LIN {X 0,Y 405.871,Z 975.986,A -85,B 0,C 180,E1 10185.137,E2 10185.137} C_VEL
LIN {X 0,Y 407.952,Z 961.068,A -85,B 0,C 180,E1 10190.645,E2 10190.645} C_VEL
LIN {X 0,Y 411.972,Z 940.342,A -85,B 0,C 180,E1 10196.169,E2 10196.169} C_VEL
LIN {X 0,Y 417.617,Z 915.19,A -85,B 0,C 180,E1 10201.176,E2 10201.176} C_VEL
LIN {X 0,Y 424.499,Z 886.002,A -85,B 0,C 180,E1 10205.579,E2 10205.579} C_VEL
LIN {X 0,Y 432.002,Z 852.461,A -85,B 0,C 180,E1 10209.402,E2 10209.402} C_VEL
LIN {X 0,Y 439.513,Z 814.318,A -85,B 0,C 180,E1 10212.598,E2 10212.598} C_VEL
LIN {X 0,Y 446.008,Z 773.682,A -85,B 0,C 180,E1 10214.978,E2 10214.978} C_VEL
LIN {X 0,Y 444.947,Z 768.035,A -85,B 0,C 180,E1 10215.473,E2 10215.473} C_VEL
LIN {X 0,Y 431.141,Z 737.427,A -85,B 0,C 180,E1 10219.164,E2 10219.164} C_VEL
LIN {X 0,Y 414.149,Z 709.31,A -85,B 0,C 180,E1 10223.192,E2 10223.192} C_VEL
LIN {X 0,Y 406.063,Z 697.489,A -85,B 0,C 180,E1 10225.147,E2 10225.147} C_VEL
LIN {X 0,Y 403.307,Z 692.479,A -85,B 0,C 180,E1 10225.876,E2 10225.876} C_VEL
LIN {X 0,Y 403.251,Z 691.44,A -85,B 0,C 180,E1 10226.097,E2 10226.097} C_VEL
LIN {X 0,Y 403.428,Z 691.44,A -85,B 0,C 180,E1 10233.243,E2 10233.243} C_VEL
LIN {X 0,Y 403.698,Z 691.44,A -85,B 0,C 180,E1 10240.281,E2 10240.281} C_VEL
LIN {X 0,Y 403.994,Z 691.44,A -85,B 0,C 180,E1 10247.012,E2 10247.012} C_VEL
LIN {X 0,Y 404.187,Z 691.44,A -85,B 0,C 180,E1 10253.554,E2 10253.554} C_VEL
LIN {X 0,Y 404.547,Z 691.44,A -85,B 0,C 180,E1 10260.005,E2 10260.005} C_VEL
LIN {X 0,Y 404.199,Z 691.44,A -85,B 0,C 180,E1 10266.457,E2 10266.457} C_VEL
LIN {X 0,Y 403.89,Z 691.44,A -85,B 0,C 180,E1 10273.002,E2 10273.002} C_VEL
LIN {X 0,Y 403.653,Z 691.44,A -85,B 0,C 180,E1 10279.732,E2 10279.732} C_VEL
LIN {X 0,Y 403.436,Z 691.44,A -85,B 0,C 180,E1 10286.768,E2 10286.768} C_VEL
LIN {X 0,Y 403.325,Z 692.074,A -85,B 0,C 180,E1 10293.543,E2 10293.543} C_VEL
LIN {X 0,Y 405.891,Z 697.335,A -85,B 0,C 180,E1 10294.241,E2 10294.241} C_VEL
LIN {X 0,Y 408.427,Z 700.839,A -85,B 0,C 180,E1 10294.859,E2 10294.859} C_VEL
LIN {X 0,Y 427.36,Z 729.308,A -85,B 0,C 180,E1 10299.089,E2 10299.089} C_VEL
LIN {X 0,Y 444.306,Z 761.012,A -85,B 0,C 180,E1 10302.797,E2 10302.797} C_VEL
LIN {X 0,Y 448.42,Z 772.307,A -85,B 0,C 180,E1 10303.868,E2 10303.868} C_VEL
LIN {X 0,Y 442.82,Z 814.858,A -85,B 0,C 180,E1 10305.797,E2 10305.797} C_VEL
LIN {X 0,Y 435.789,Z 854.926,A -85,B 0,C 180,E1 10308.487,E2 10308.487} C_VEL
LIN {X 0,Y 427.875,Z 893.059,A -85,B 0,C 180,E1 10312.061,E2 10312.061} C_VEL
LIN {X 0,Y 420.295,Z 927.543,A -85,B 0,C 180,E1 10316.454,E2 10316.454} C_VEL
LIN {X 0,Y 413.816,Z 957.71,A -85,B 0,C 180,E1 10321.599,E2 10321.599} C_VEL
LIN {X 0,Y 409.877,Z 978.091,A -85,B 0,C 180,E1 10326.142,E2 10326.142} C_VEL
LIN {X 0,Y 407.965,Z 982.373,A -85,B 0,C 180,E1 10327.183,E2 10327.183} C_VEL
LIN {X 0,Y 399.703,Z 993.008,A -85,B 0,C 180,E1 10330.043,E2 10330.043} C_VEL
LIN {X 0,Y 399.497,Z 993.911,A -85,B 0,C 180,E1 10330.327,E2 10330.327} C_VEL
LIN {X 0,Y 397.623,Z 1008.916,A -85,B 0,C 180,E1 10336.293,E2 10336.293} C_VEL
LIN {X 0,Y 397.001,Z 1017.213,A -85,B 0,C 180,E1 10341.226,E2 10341.226} C_VEL
LIN {X 0,Y 396.743,Z 1021.482,A -85,B 0,C 180,E1 10345.623,E2 10345.623} C_VEL
LIN {X 0,Y 396.752,Z 1022.899,A -85,B 0,C 180,E1 10350,E2 10350} C_VEL
LIN {X 0,Y 396.734,Z 1021.482,A -85,B 0,C 180,E1 10354.378,E2 10354.378} C_VEL
LIN {X 0,Y 397.07,Z 1015.608,A -85,B 0,C 180,E1 10359.881,E2 10359.881} C_VEL
LIN {X 0,Y 398.017,Z 1005.17,A -85,B 0,C 180,E1 10365.444,E2 10365.444} C_VEL
LIN {X 0,Y 400.499,Z 987.673,A -85,B 0,C 180,E1 10371.63,E2 10371.63} C_VEL
LIN {X 0,Y 405.041,Z 964.149,A -85,B 0,C 180,E1 10377.555,E2 10377.555} C_VEL
LIN {X 0,Y 411.393,Z 936.262,A -85,B 0,C 180,E1 10382.768,E2 10382.768} C_VEL
LIN {X 0,Y 419.069,Z 903.077,A -85,B 0,C 180,E1 10387.428,E2 10387.428} C_VEL
LIN {X 0,Y 427.424,Z 865.851,A -85,B 0,C 180,E1 10391.282,E2 10391.282} C_VEL
LIN {X 0,Y 435.091,Z 826.33,A -85,B 0,C 180,E1 10394.246,E2 10394.246} C_VEL
LIN {X 0,Y 441.567,Z 783.435,A -85,B 0,C 180,E1 10396.448,E2 10396.448} C_VEL
LIN {X 0,Y 442.358,Z 773.084,A -85,B 0,C 180,E1 10396.899,E2 10396.899} C_VEL
LIN {X 0,Y 427.471,Z 742.287,A -85,B 0,C 180,E1 10400.473,E2 10400.473} C_VEL
LIN {X 0,Y 410.7,Z 715.445,A -85,B 0,C 180,E1 10404.281,E2 10404.281} C_VEL
LIN {X 0,Y 398.509,Z 697.759,A -85,B 0,C 180,E1 10407.342,E2 10407.342} C_VEL
LIN {X 0,Y 395.501,Z 692.766,A -85,B 0,C 180,E1 10408.189,E2 10408.189} C_VEL
LIN {X 0,Y 395.382,Z 691.44,A -85,B 0,C 180,E1 10408.316,E2 10408.316} C_VEL
LIN {X 0,Y 395.521,Z 691.44,A -85,B 0,C 180,E1 10415.095,E2 10415.095} C_VEL
LIN {X 0,Y 395.755,Z 691.44,A -85,B 0,C 180,E1 10422.175,E2 10422.175} C_VEL
LIN {X 0,Y 395.918,Z 691.44,A -85,B 0,C 180,E1 10428.973,E2 10428.973} C_VEL
LIN {X 0,Y 396.325,Z 691.44,A -85,B 0,C 180,E1 10435.613,E2 10435.613} C_VEL
LIN {X 0,Y 396.584,Z 691.44,A -85,B 0,C 180,E1 10439.995,E2 10439.995} C_VEL
LIN {X 0,Y 396.272,Z 691.44,A -85,B 0,C 180,E1 10446.576,E2 10446.576} C_VEL
LIN {X 0,Y 395.972,Z 691.44,A -85,B 0,C 180,E1 10453.256,E2 10453.256} C_VEL
LIN {X 0,Y 395.763,Z 691.44,A -85,B 0,C 180,E1 10460.131,E2 10460.131} C_VEL
LIN {X 0,Y 395.465,Z 691.44,A -85,B 0,C 180,E1 10467.34,E2 10467.34} C_VEL
LIN {X 0,Y 395.414,Z 691.44,A -85,B 0,C 180,E1 10472.224,E2 10472.224} C_VEL
LIN {X 0,Y 397.431,Z 696.7,A -85,B 0,C 180,E1 10472.865,E2 10472.865} C_VEL
LIN {X 0,Y 400.544,Z 700.599,A -85,B 0,C 180,E1 10473.678,E2 10473.678} C_VEL
LIN {X 0,Y 416.344,Z 724.657,A -85,B 0,C 180,E1 10477.679,E2 10477.679} C_VEL
LIN {X 0,Y 431.961,Z 754.146,A -85,B 0,C 180,E1 10481.744,E2 10481.744} C_VEL
LIN {X 0,Y 440.414,Z 774.599,A -85,B 0,C 180,E1 10484.234,E2 10484.234} C_VEL
LIN {X 0,Y 433.168,Z 817.314,A -85,B 0,C 180,E1 10486.78,E2 10486.78} C_VEL
LIN {X 0,Y 425.102,Z 855.93,A -85,B 0,C 180,E1 10490.125,E2 10490.125} C_VEL
LIN {X 0,Y 417.01,Z 890.098,A -85,B 0,C 180,E1 10494.18,E2 10494.18} C_VEL
LIN {X 0,Y 409.351,Z 920.988,A -85,B 0,C 180,E1 10499.122,E2 10499.122} C_VEL
LIN {X 0,Y 403.241,Z 947.182,A -85,B 0,C 180,E1 10504.818,E2 10504.818} C_VEL
LIN {X 0,Y 399.451,Z 967.283,A -85,B 0,C 180,E1 10510.858,E2 10510.858} C_VEL
LIN {X 0,Y 397.531,Z 981.028,A -85,B 0,C 180,E1 10516.789,E2 10516.789} C_VEL
LIN {X 0,Y 396.87,Z 989.319,A -85,B 0,C 180,E1 10522.606,E2 10522.606} C_VEL
LIN {X 0,Y 396.723,Z 992.824,A -85,B 0,C 180,E1 10527.812,E2 10527.812} C_VEL
LIN {X 0,Y 396.715,Z 992.797,A -85,B 0,C 180,E1 10532.187,E2 10532.187} C_VEL
LIN {X 0,Y 396.85,Z 989.248,A -85,B 0,C 180,E1 10537.371,E2 10537.371} C_VEL
LIN {X 0,Y 397.582,Z 980.849,A -85,B 0,C 180,E1 10543.208,E2 10543.208} C_VEL
LIN {X 0,Y 399.731,Z 965.902,A -85,B 0,C 180,E1 10549.543,E2 10549.543} C_VEL
LIN {X 0,Y 403.525,Z 945.764,A -85,B 0,C 180,E1 10555.461,E2 10555.461} C_VEL
LIN {X 0,Y 409.55,Z 920.56,A -85,B 0,C 180,E1 10560.86,E2 10560.86} C_VEL
LIN {X 0,Y 417.157,Z 889.469,A -85,B 0,C 180,E1 10565.813,E2 10565.813} C_VEL
LIN {X 0,Y 425.282,Z 855.209,A -85,B 0,C 180,E1 10569.854,E2 10569.854} C_VEL
LIN {X 0,Y 433.349,Z 816.503,A -85,B 0,C 180,E1 10573.181,E2 10573.181} C_VEL
LIN {X 0,Y 440.244,Z 774.615,A -85,B 0,C 180,E1 10575.694,E2 10575.694} C_VEL
LIN {X 0,Y 427.49,Z 744.686,A -85,B 0,C 180,E1 10579.381,E2 10579.381} C_VEL
LIN {X 0,Y 410.721,Z 715.714,A -85,B 0,C 180,E1 10583.622,E2 10583.622} C_VEL
LIN {X 0,Y 398.207,Z 697.529,A -85,B 0,C 180,E1 10586.822,E2 10586.822} C_VEL
LIN {X 0,Y 395.46,Z 692.854,A -85,B 0,C 180,E1 10587.599,E2 10587.599} C_VEL
LIN {X 0,Y 395.322,Z 691.44,A -85,B 0,C 180,E1 10587.77,E2 10587.77} C_VEL
LIN {X 0,Y 395.539,Z 691.44,A -85,B 0,C 180,E1 10595.107,E2 10595.107} C_VEL
LIN {X 0,Y 395.888,Z 691.44,A -85,B 0,C 180,E1 10602.192,E2 10602.192} C_VEL
LIN {X 0,Y 396.138,Z 691.44,A -85,B 0,C 180,E1 10608.99,E2 10608.99} C_VEL
LIN {X 0,Y 396.441,Z 691.44,A -85,B 0,C 180,E1 10615.625,E2 10615.625} C_VEL
LIN {X 0,Y 396.615,Z 691.44,A -85,B 0,C 180,E1 10622.193,E2 10622.193} C_VEL
LIN {X 0,Y 396.164,Z 691.44,A -85,B 0,C 180,E1 10628.798,E2 10628.798} C_VEL
LIN {X 0,Y 395.869,Z 691.44,A -85,B 0,C 180,E1 10635.532,E2 10635.532} C_VEL
LIN {X 0,Y 395.623,Z 691.44,A -85,B 0,C 180,E1 10642.504,E2 10642.504} C_VEL
LIN {X 0,Y 395.397,Z 691.44,A -85,B 0,C 180,E1 10649.856,E2 10649.856} C_VEL
LIN {X 0,Y 395.38,Z 691.837,A -85,B 0,C 180,E1 10651.776,E2 10651.776} C_VEL
LIN {X 0,Y 397.682,Z 697.026,A -85,B 0,C 180,E1 10652.472,E2 10652.472} C_VEL
LIN {X 0,Y 400.23,Z 700.075,A -85,B 0,C 180,E1 10653.132,E2 10653.132} C_VEL
LIN {X 0,Y 420.31,Z 729.973,A -85,B 0,C 180,E1 10657.926,E2 10657.926} C_VEL
LIN {X 0,Y 437.407,Z 761.803,A -85,B 0,C 180,E1 10661.868,E2 10661.868} C_VEL
LIN {X 0,Y 442.611,Z 774.779,A -85,B 0,C 180,E1 10663.231,E2 10663.231} C_VEL
LIN {X 0,Y 436.936,Z 815.44,A -85,B 0,C 180,E1 10665.114,E2 10665.114} C_VEL
LIN {X 0,Y 429.605,Z 855.135,A -85,B 0,C 180,E1 10667.809,E2 10667.809} C_VEL
LIN {X 0,Y 421.323,Z 893.161,A -85,B 0,C 180,E1 10671.421,E2 10671.421} C_VEL
LIN {X 0,Y 413.286,Z 927.882,A -85,B 0,C 180,E1 10675.923,E2 10675.923} C_VEL
LIN {X 0,Y 406.574,Z 957.4,A -85,B 0,C 180,E1 10681.046,E2 10681.046} C_VEL
LIN {X 0,Y 401.645,Z 981.707,A -85,B 0,C 180,E1 10686.683,E2 10686.683} C_VEL
LIN {X 0,Y 399.497,Z 993.911,A -85,B 0,C 180,E1 10690.327,E2 10690.327} C_VEL
LIN {X 0,Y 396.338,Z 999.066,A -85,B 0,C 180,E1 10692.008,E2 10692.008} C_VEL
LIN {X 0,Y 390.178,Z 1005.669,A -85,B 0,C 180,E1 10694.591,E2 10694.591} C_VEL
LIN {X 0,Y 390.011,Z 1006.311,A -85,B 0,C 180,E1 10694.899,E2 10694.899} C_VEL
LIN {X 0,Y 389.097,Z 1016.913,A -85,B 0,C 180,E1 10701.046,E2 10701.046} C_VEL
LIN {X 0,Y 388.839,Z 1021.185,A -85,B 0,C 180,E1 10705.534,E2 10705.534} C_VEL
LIN {X 0,Y 388.883,Z 1022.604,A -85,B 0,C 180,E1 10710,E2 10710} C_VEL
LIN {X 0,Y 388.831,Z 1021.185,A -85,B 0,C 180,E1 10714.467,E2 10714.467} C_VEL
LIN {X 0,Y 389.187,Z 1015.307,A -85,B 0,C 180,E1 10720.083,E2 10720.083} C_VEL
LIN {X 0,Y 390.208,Z 1004.866,A -85,B 0,C 180,E1 10725.761,E2 10725.761} C_VEL
LIN {X 0,Y 392.769,Z 987.927,A -85,B 0,C 180,E1 10731.907,E2 10731.907} C_VEL
LIN {X 0,Y 397.603,Z 964.446,A -85,B 0,C 180,E1 10737.977,E2 10737.977} C_VEL
LIN {X 0,Y 404.532,Z 935.531,A -85,B 0,C 180,E1 10743.472,E2 10743.472} C_VEL
LIN {X 0,Y 412.644,Z 902.628,A -85,B 0,C 180,E1 10748.135,E2 10748.135} C_VEL
LIN {X 0,Y 421.305,Z 865.723,A -85,B 0,C 180,E1 10751.998,E2 10751.998} C_VEL
LIN {X 0,Y 429.393,Z 825.785,A -85,B 0,C 180,E1 10755.012,E2 10755.012} C_VEL
LIN {X 0,Y 436.114,Z 783.096,A -85,B 0,C 180,E1 10757.21,E2 10757.21} C_VEL
LIN {X 0,Y 436.335,Z 775.895,A -85,B 0,C 180,E1 10757.577,E2 10757.577} C_VEL
LIN {X 0,Y 422.102,Z 745.957,A -85,B 0,C 180,E1 10761.2,E2 10761.2} C_VEL
LIN {X 0,Y 404.297,Z 717.07,A -85,B 0,C 180,E1 10765.501,E2 10765.501} C_VEL
LIN {X 0,Y 394.117,Z 702.978,A -85,B 0,C 180,E1 10768.167,E2 10768.167} C_VEL
LIN {X 0,Y 390.792,Z 697.897,A -85,B 0,C 180,E1 10769.13,E2 10769.13} C_VEL
LIN {X 0,Y 387.726,Z 693.299,A -85,B 0,C 180,E1 10770.055,E2 10770.055} C_VEL
LIN {X 0,Y 387.494,Z 691.44,A -85,B 0,C 180,E1 10770.29,E2 10770.29} C_VEL
LIN {X 0,Y 387.666,Z 691.44,A -85,B 0,C 180,E1 10777.008,E2 10777.008} C_VEL
LIN {X 0,Y 387.84,Z 691.44,A -85,B 0,C 180,E1 10784.138,E2 10784.138} C_VEL
LIN {X 0,Y 388.185,Z 691.44,A -85,B 0,C 180,E1 10791.02,E2 10791.02} C_VEL
LIN {X 0,Y 388.714,Z 691.44,A -85,B 0,C 180,E1 10797.763,E2 10797.763} C_VEL
LIN {X 0,Y 388.477,Z 691.44,A -85,B 0,C 180,E1 10804.465,E2 10804.465} C_VEL
LIN {X 0,Y 388.114,Z 691.44,A -85,B 0,C 180,E1 10811.241,E2 10811.241} C_VEL
LIN {X 0,Y 387.896,Z 691.44,A -85,B 0,C 180,E1 10818.188,E2 10818.188} C_VEL
LIN {X 0,Y 387.566,Z 691.44,A -85,B 0,C 180,E1 10825.441,E2 10825.441} C_VEL
LIN {X 0,Y 387.513,Z 691.604,A -85,B 0,C 180,E1 10830.313,E2 10830.313} C_VEL
LIN {X 0,Y 389.444,Z 696.62,A -85,B 0,C 180,E1 10830.978,E2 10830.978} C_VEL
LIN {X 0,Y 392.499,Z 700,A -85,B 0,C 180,E1 10831.835,E2 10831.835} C_VEL
LIN {X 0,Y 409.2,Z 725.217,A -85,B 0,C 180,E1 10836.37,E2 10836.37} C_VEL
LIN {X 0,Y 424.361,Z 753.408,A -85,B 0,C 180,E1 10840.51,E2 10840.51} C_VEL
LIN {X 0,Y 434.373,Z 777.629,A -85,B 0,C 180,E1 10843.602,E2 10843.602} C_VEL
LIN {X 0,Y 427.137,Z 818.664,A -85,B 0,C 180,E1 10846.124,E2 10846.124} C_VEL
LIN {X 0,Y 418.893,Z 856.23,A -85,B 0,C 180,E1 10849.412,E2 10849.412} C_VEL
LIN {X 0,Y 410.389,Z 890.63,A -85,B 0,C 180,E1 10853.549,E2 10853.549} C_VEL
LIN {X 0,Y 402.372,Z 921.29,A -85,B 0,C 180,E1 10858.526,E2 10858.526} C_VEL
LIN {X 0,Y 396.111,Z 946.646,A -85,B 0,C 180,E1 10864.093,E2 10864.093} C_VEL
LIN {X 0,Y 391.859,Z 967.323,A -85,B 0,C 180,E1 10870.37,E2 10870.37} C_VEL
LIN {X 0,Y 389.739,Z 981.327,A -85,B 0,C 180,E1 10876.52,E2 10876.52} C_VEL
LIN {X 0,Y 388.984,Z 989.616,A -85,B 0,C 180,E1 10882.455,E2 10882.455} C_VEL
LIN {X 0,Y 388.83,Z 993.12,A -85,B 0,C 180,E1 10887.768,E2 10887.768} C_VEL
LIN {X 0,Y 388.82,Z 993.094,A -85,B 0,C 180,E1 10892.231,E2 10892.231} C_VEL
LIN {X 0,Y 388.964,Z 989.547,A -85,B 0,C 180,E1 10897.521,E2 10897.521} C_VEL
LIN {X 0,Y 389.798,Z 981.15,A -85,B 0,C 180,E1 10903.477,E2 10903.477} C_VEL
LIN {X 0,Y 391.954,Z 967.034,A -85,B 0,C 180,E1 10909.648,E2 10909.648} C_VEL
LIN {X 0,Y 396.14,Z 946.287,A -85,B 0,C 180,E1 10915.915,E2 10915.915} C_VEL
LIN {X 0,Y 402.524,Z 920.874,A -85,B 0,C 180,E1 10921.459,E2 10921.459} C_VEL
LIN {X 0,Y 410.549,Z 890.02,A -85,B 0,C 180,E1 10926.443,E2 10926.443} C_VEL
LIN {X 0,Y 419.131,Z 855.517,A -85,B 0,C 180,E1 10930.559,E2 10930.559} C_VEL
LIN {X 0,Y 427.707,Z 816.033,A -85,B 0,C 180,E1 10933.967,E2 10933.967} C_VEL
LIN {X 0,Y 434.276,Z 777.765,A -85,B 0,C 180,E1 10936.306,E2 10936.306} C_VEL
LIN {X 0,Y 421.778,Z 747.945,A -85,B 0,C 180,E1 10940.144,E2 10940.144} C_VEL
LIN {X 0,Y 406.249,Z 720.645,A -85,B 0,C 180,E1 10944.315,E2 10944.315} C_VEL
LIN {X 0,Y 394.627,Z 703.593,A -85,B 0,C 180,E1 10947.432,E2 10947.432} C_VEL
LIN {X 0,Y 390.66,Z 697.774,A -85,B 0,C 180,E1 10948.567,E2 10948.567} C_VEL
LIN {X 0,Y 387.611,Z 692.986,A -85,B 0,C 180,E1 10949.493,E2 10949.493} C_VEL
LIN {X 0,Y 387.439,Z 691.44,A -85,B 0,C 180,E1 10949.682,E2 10949.682} C_VEL
LIN {X 0,Y 387.675,Z 691.44,A -85,B 0,C 180,E1 10957.02,E2 10957.02} C_VEL
LIN {X 0,Y 388.036,Z 691.44,A -85,B 0,C 180,E1 10964.157,E2 10964.157} C_VEL
LIN {X 0,Y 388.261,Z 691.44,A -85,B 0,C 180,E1 10971.233,E2 10971.233} C_VEL
LIN {X 0,Y 388.66,Z 691.44,A -85,B 0,C 180,E1 10977.773,E2 10977.773} C_VEL
LIN {X 0,Y 388.721,Z 691.44,A -85,B 0,C 180,E1 10982.237,E2 10982.237} C_VEL
LIN {X 0,Y 388.225,Z 691.44,A -85,B 0,C 180,E1 10988.979,E2 10988.979} C_VEL
LIN {X 0,Y 387.956,Z 691.44,A -85,B 0,C 180,E1 10995.858,E2 10995.858} C_VEL
LIN {X 0,Y 387.676,Z 691.44,A -85,B 0,C 180,E1 11002.991,E2 11002.991} C_VEL
LIN {X 0,Y 387.509,Z 691.752,A -85,B 0,C 180,E1 11009.864,E2 11009.864} C_VEL
LIN {X 0,Y 389.61,Z 696.874,A -85,B 0,C 180,E1 11010.572,E2 11010.572} C_VEL
LIN {X 0,Y 392.432,Z 699.946,A -85,B 0,C 180,E1 11011.36,E2 11011.36} C_VEL
LIN {X 0,Y 410.252,Z 726.239,A -85,B 0,C 180,E1 11015.98,E2 11015.98} C_VEL
LIN {X 0,Y 426.337,Z 753.807,A -85,B 0,C 180,E1 11019.818,E2 11019.818} C_VEL
LIN {X 0,Y 436.774,Z 777.147,A -85,B 0,C 180,E1 11022.559,E2 11022.559} C_VEL
LIN {X 0,Y 430.955,Z 816.904,A -85,B 0,C 180,E1 11024.464,E2 11024.464} C_VEL
LIN {X 0,Y 423.306,Z 856.219,A -85,B 0,C 180,E1 11027.189,E2 11027.189} C_VEL
LIN {X 0,Y 414.761,Z 893.451,A -85,B 0,C 180,E1 11030.781,E2 11030.781} C_VEL
LIN {X 0,Y 406.466,Z 927.503,A -85,B 0,C 180,E1 11035.258,E2 11035.258} C_VEL
LIN {X 0,Y 399.337,Z 957.089,A -85,B 0,C 180,E1 11040.47,E2 11040.47} C_VEL
LIN {X 0,Y 394.118,Z 981.399,A -85,B 0,C 180,E1 11046.211,E2 11046.211} C_VEL
LIN {X 0,Y 390.795,Z 1000.752,A -85,B 0,C 180,E1 11052.527,E2 11052.527} C_VEL
LIN {X 0,Y 390.011,Z 1006.311,A -85,B 0,C 180,E1 11054.899,E2 11054.899} C_VEL
LIN {X 0,Y 387.127,Z 1010.096,A -85,B 0,C 180,E1 11056.708,E2 11056.708} C_VEL
LIN {X 0,Y 381.403,Z 1014.666,A -85,B 0,C 180,E1 11059.46,E2 11059.46} C_VEL
LIN {X 0,Y 381.271,Z 1015.113,A -85,B 0,C 180,E1 11059.783,E2 11059.783} C_VEL
LIN {X 0,Y 380.936,Z 1020.888,A -85,B 0,C 180,E1 11065.441,E2 11065.441} C_VEL
LIN {X 0,Y 380.987,Z 1022.308,A -85,B 0,C 180,E1 11070,E2 11070} C_VEL
LIN {X 0,Y 380.927,Z 1020.888,A -85,B 0,C 180,E1 11074.56,E2 11074.56} C_VEL
LIN {X 0,Y 381.312,Z 1015.007,A -85,B 0,C 180,E1 11080.293,E2 11080.293} C_VEL
LIN {X 0,Y 382.409,Z 1004.561,A -85,B 0,C 180,E1 11086.091,E2 11086.091} C_VEL
LIN {X 0,Y 385.08,Z 988,A -85,B 0,C 180,E1 11092.241,E2 11092.241} C_VEL
LIN {X 0,Y 390.246,Z 964.424,A -85,B 0,C 180,E1 11098.483,E2 11098.483} C_VEL
LIN {X 0,Y 397.61,Z 935.371,A -85,B 0,C 180,E1 11104.106,E2 11104.106} C_VEL
LIN {X 0,Y 406.391,Z 901.628,A -85,B 0,C 180,E1 11108.933,E2 11108.933} C_VEL
LIN {X 0,Y 415.124,Z 866.198,A -85,B 0,C 180,E1 11112.681,E2 11112.681} C_VEL
LIN {X 0,Y 423.372,Z 827.365,A -85,B 0,C 180,E1 11115.664,E2 11115.664} C_VEL
LIN {X 0,Y 430.534,Z 784.272,A -85,B 0,C 180,E1 11117.93,E2 11117.93} C_VEL
LIN {X 0,Y 430.282,Z 778.38,A -85,B 0,C 180,E1 11118.306,E2 11118.306} C_VEL
LIN {X 0,Y 416.342,Z 748.795,A -85,B 0,C 180,E1 11122.061,E2 11122.061} C_VEL
LIN {X 0,Y 399.171,Z 720.875,A -85,B 0,C 180,E1 11126.456,E2 11126.456} C_VEL
LIN {X 0,Y 387.074,Z 703.849,A -85,B 0,C 180,E1 11129.84,E2 11129.84} C_VEL
LIN {X 0,Y 383.005,Z 697.964,A -85,B 0,C 180,E1 11131.115,E2 11131.115} C_VEL
LIN {X 0,Y 379.872,Z 693.418,A -85,B 0,C 180,E1 11132.153,E2 11132.153} C_VEL
LIN {X 0,Y 379.605,Z 691.44,A -85,B 0,C 180,E1 11132.374,E2 11132.374} C_VEL
LIN {X 0,Y 379.797,Z 691.44,A -85,B 0,C 180,E1 11138.971,E2 11138.971} C_VEL
LIN {X 0,Y 379.931,Z 691.44,A -85,B 0,C 180,E1 11146.162,E2 11146.162} C_VEL
LIN {X 0,Y 380.438,Z 691.44,A -85,B 0,C 180,E1 11153.138,E2 11153.138} C_VEL
LIN {X 0,Y 380.79,Z 691.44,A -85,B 0,C 180,E1 11159.994,E2 11159.994} C_VEL
LIN {X 0,Y 380.437,Z 691.44,A -85,B 0,C 180,E1 11166.851,E2 11166.851} C_VEL
LIN {X 0,Y 380.102,Z 691.44,A -85,B 0,C 180,E1 11173.82,E2 11173.82} C_VEL
LIN {X 0,Y 379.827,Z 691.44,A -85,B 0,C 180,E1 11181.015,E2 11181.015} C_VEL
LIN {X 0,Y 379.654,Z 691.44,A -85,B 0,C 180,E1 11188.175,E2 11188.175} C_VEL
LIN {X 0,Y 381.526,Z 696.61,A -85,B 0,C 180,E1 11188.915,E2 11188.915} C_VEL
LIN {X 0,Y 384.734,Z 700.036,A -85,B 0,C 180,E1 11189.903,E2 11189.903} C_VEL
LIN {X 0,Y 401.207,Z 724.075,A -85,B 0,C 180,E1 11194.711,E2 11194.711} C_VEL
LIN {X 0,Y 417.592,Z 754.476,A -85,B 0,C 180,E1 11199.454,E2 11199.454} C_VEL
LIN {X 0,Y 428.42,Z 780.825,A -85,B 0,C 180,E1 11202.984,E2 11202.984} C_VEL
LIN {X 0,Y 421.258,Z 819.645,A -85,B 0,C 180,E1 11205.424,E2 11205.424} C_VEL
LIN {X 0,Y 412.809,Z 856.527,A -85,B 0,C 180,E1 11208.685,E2 11208.685} C_VEL
LIN {X 0,Y 403.874,Z 891.026,A -85,B 0,C 180,E1 11212.88,E2 11212.88} C_VEL
LIN {X 0,Y 395.428,Z 921.593,A -85,B 0,C 180,E1 11217.908,E2 11217.908} C_VEL
LIN {X 0,Y 388.827,Z 946.909,A -85,B 0,C 180,E1 11223.559,E2 11223.559} C_VEL
LIN {X 0,Y 384.285,Z 967.226,A -85,B 0,C 180,E1 11229.807,E2 11229.807} C_VEL
LIN {X 0,Y 381.946,Z 981.626,A -85,B 0,C 180,E1 11236.24,E2 11236.24} C_VEL
LIN {X 0,Y 381.12,Z 989.616,A -85,B 0,C 180,E1 11242.007,E2 11242.007} C_VEL
LIN {X 0,Y 380.931,Z 993.416,A -85,B 0,C 180,E1 11247.722,E2 11247.722} C_VEL
LIN {X 0,Y 380.92,Z 993.39,A -85,B 0,C 180,E1 11252.278,E2 11252.278} C_VEL
LIN {X 0,Y 381.106,Z 989.524,A -85,B 0,C 180,E1 11257.992,E2 11257.992} C_VEL
LIN {X 0,Y 382.127,Z 980.528,A -85,B 0,C 180,E1 11264.237,E2 11264.237} C_VEL
LIN {X 0,Y 384.349,Z 966.958,A -85,B 0,C 180,E1 11270.201,E2 11270.201} C_VEL
LIN {X 0,Y 388.865,Z 946.539,A -85,B 0,C 180,E1 11276.452,E2 11276.452} C_VEL
LIN {X 0,Y 395.553,Z 921.183,A -85,B 0,C 180,E1 11282.08,E2 11282.08} C_VEL
LIN {X 0,Y 404.058,Z 890.442,A -85,B 0,C 180,E1 11287.107,E2 11287.107} C_VEL
LIN {X 0,Y 413.042,Z 855.824,A -85,B 0,C 180,E1 11291.286,E2 11291.286} C_VEL
LIN {X 0,Y 421.819,Z 817.265,A -85,B 0,C 180,E1 11294.655,E2 11294.655} C_VEL
LIN {X 0,Y 428.325,Z 780.971,A -85,B 0,C 180,E1 11296.923,E2 11296.923} C_VEL
LIN {X 0,Y 416.664,Z 752.449,A -85,B 0,C 180,E1 11300.732,E2 11300.732} C_VEL
LIN {X 0,Y 400.891,Z 723.831,A -85,B 0,C 180,E1 11305.258,E2 11305.258} C_VEL
LIN {X 0,Y 387.309,Z 704.154,A -85,B 0,C 180,E1 11309.168,E2 11309.168} C_VEL
LIN {X 0,Y 382.938,Z 697.914,A -85,B 0,C 180,E1 11310.53,E2 11310.53} C_VEL
LIN {X 0,Y 379.762,Z 693.059,A -85,B 0,C 180,E1 11311.59,E2 11311.59} C_VEL
LIN {X 0,Y 379.593,Z 691.44,A -85,B 0,C 180,E1 11311.739,E2 11311.739} C_VEL
LIN {X 0,Y 379.827,Z 691.44,A -85,B 0,C 180,E1 11318.985,E2 11318.985} C_VEL
LIN {X 0,Y 380.163,Z 691.44,A -85,B 0,C 180,E1 11326.182,E2 11326.182} C_VEL
LIN {X 0,Y 380.469,Z 691.44,A -85,B 0,C 180,E1 11333.15,E2 11333.15} C_VEL
LIN {X 0,Y 380.849,Z 691.44,A -85,B 0,C 180,E1 11340.006,E2 11340.006} C_VEL
LIN {X 0,Y 380.437,Z 691.44,A -85,B 0,C 180,E1 11346.862,E2 11346.862} C_VEL
LIN {X 0,Y 380.084,Z 691.44,A -85,B 0,C 180,E1 11353.832,E2 11353.832} C_VEL
LIN {X 0,Y 379.797,Z 691.44,A -85,B 0,C 180,E1 11361.029,E2 11361.029} C_VEL
LIN {X 0,Y 379.679,Z 692.237,A -85,B 0,C 180,E1 11367.782,E2 11367.782} C_VEL
LIN {X 0,Y 382.284,Z 697.399,A -85,B 0,C 180,E1 11368.702,E2 11368.702} C_VEL
LIN {X 0,Y 384.769,Z 700.188,A -85,B 0,C 180,E1 11369.466,E2 11369.466} C_VEL
LIN {X 0,Y 402.141,Z 725.186,A -85,B 0,C 180,E1 11374.338,E2 11374.338} C_VEL
LIN {X 0,Y 418.613,Z 753.04,A -85,B 0,C 180,E1 11378.52,E2 11378.52} C_VEL
LIN {X 0,Y 431.025,Z 780.4,A -85,B 0,C 180,E1 11381.924,E2 11381.924} C_VEL
LIN {X 0,Y 424.703,Z 820.098,A -85,B 0,C 180,E1 11383.898,E2 11383.898} C_VEL
LIN {X 0,Y 416.988,Z 857.539,A -85,B 0,C 180,E1 11386.568,E2 11386.568} C_VEL
LIN {X 0,Y 408.27,Z 893.853,A -85,B 0,C 180,E1 11390.139,E2 11390.139} C_VEL
LIN {X 0,Y 399.626,Z 927.5,A -85,B 0,C 180,E1 11394.632,E2 11394.632} C_VEL
LIN {X 0,Y 392.191,Z 956.779,A -85,B 0,C 180,E1 11399.876,E2 11399.876} C_VEL
LIN {X 0,Y 386.55,Z 981.089,A -85,B 0,C 180,E1 11405.715,E2 11405.715} C_VEL
LIN {X 0,Y 383.06,Z 1000.447,A -85,B 0,C 180,E1 11412.162,E2 11412.162} C_VEL
LIN {X 0,Y 381.402,Z 1013.369,A -85,B 0,C 180,E1 11418.552,E2 11418.552} C_VEL
LIN {X 0,Y 381.271,Z 1015.113,A -85,B 0,C 180,E1 11419.783,E2 11419.783} C_VEL
LIN {X 0,Y 378.543,Z 1017.527,A -85,B 0,C 180,E1 11421.689,E2 11421.689} C_VEL
LIN {X 0,Y 373.113,Z 1020.025,A -85,B 0,C 180,E1 11424.585,E2 11424.585} C_VEL
LIN {X 0,Y 373.033,Z 1020.27,A -85,B 0,C 180,E1 11424.921,E2 11424.921} C_VEL
LIN {X 0,Y 373.116,Z 1022.013,A -85,B 0,C 180,E1 11430,E2 11430} C_VEL
LIN {X 0,Y 373.053,Z 1020.592,A -85,B 0,C 180,E1 11434.656,E2 11434.656} C_VEL
LIN {X 0,Y 373.435,Z 1014.707,A -85,B 0,C 180,E1 11440.513,E2 11440.513} C_VEL
LIN {X 0,Y 374.615,Z 1004.257,A -85,B 0,C 180,E1 11446.435,E2 11446.435} C_VEL
LIN {X 0,Y 377.774,Z 986.506,A -85,B 0,C 180,E1 11453.079,E2 11453.079} C_VEL
LIN {X 0,Y 383.001,Z 964.061,A -85,B 0,C 180,E1 11459.086,E2 11459.086} C_VEL
LIN {X 0,Y 390.905,Z 934.708,A -85,B 0,C 180,E1 11464.842,E2 11464.842} C_VEL
LIN {X 0,Y 400.054,Z 901.322,A -85,B 0,C 180,E1 11469.67,E2 11469.67} C_VEL
LIN {X 0,Y 409.368,Z 865.116,A -85,B 0,C 180,E1 11473.521,E2 11473.521} C_VEL
LIN {X 0,Y 418.101,Z 825.607,A -85,B 0,C 180,E1 11476.546,E2 11476.546} C_VEL
LIN {X 0,Y 424.913,Z 782.579,A -85,B 0,C 180,E1 11478.862,E2 11478.862} C_VEL
LIN {X 0,Y 410.894,Z 752.103,A -85,B 0,C 180,E1 11482.886,E2 11482.886} C_VEL
LIN {X 0,Y 393.642,Z 723.678,A -85,B 0,C 180,E1 11487.575,E2 11487.575} C_VEL
LIN {X 0,Y 379.978,Z 704.567,A -85,B 0,C 180,E1 11491.688,E2 11491.688} C_VEL
LIN {X 0,Y 375.6,Z 698.26,A -85,B 0,C 180,E1 11493.199,E2 11493.199} C_VEL
LIN {X 0,Y 371.973,Z 693.472,A -85,B 0,C 180,E1 11494.523,E2 11494.523} C_VEL
LIN {X 0,Y 371.693,Z 691.44,A -85,B 0,C 180,E1 11494.836,E2 11494.836} C_VEL
LIN {X 0,Y 371.926,Z 691.44,A -85,B 0,C 180,E1 11500.99,E2 11500.99} C_VEL
LIN {X 0,Y 372.104,Z 691.44,A -85,B 0,C 180,E1 11508.257,E2 11508.257} C_VEL
LIN {X 0,Y 372.602,Z 691.44,A -85,B 0,C 180,E1 11515.333,E2 11515.333} C_VEL
LIN {X 0,Y 372.889,Z 691.44,A -85,B 0,C 180,E1 11519.994,E2 11519.994} C_VEL
LIN {X 0,Y 372.51,Z 691.44,A -85,B 0,C 180,E1 11526.997,E2 11526.997} C_VEL
LIN {X 0,Y 372.159,Z 691.44,A -85,B 0,C 180,E1 11534.121,E2 11534.121} C_VEL
LIN {X 0,Y 371.851,Z 691.44,A -85,B 0,C 180,E1 11541.488,E2 11541.488} C_VEL
LIN {X 0,Y 371.777,Z 692.123,A -85,B 0,C 180,E1 11545.838,E2 11545.838} C_VEL
LIN {X 0,Y 374.22,Z 697.201,A -85,B 0,C 180,E1 11546.822,E2 11546.822} C_VEL
LIN {X 0,Y 376.998,Z 699.956,A -85,B 0,C 180,E1 11547.765,E2 11547.765} C_VEL
LIN {X 0,Y 391.99,Z 721.692,A -85,B 0,C 180,E1 11552.56,E2 11552.56} C_VEL
LIN {X 0,Y 406.986,Z 747.516,A -85,B 0,C 180,E1 11557.11,E2 11557.11} C_VEL
LIN {X 0,Y 420.206,Z 777.379,A -85,B 0,C 180,E1 11561.452,E2 11561.452} C_VEL
LIN {X 0,Y 422.569,Z 784.223,A -85,B 0,C 180,E1 11562.371,E2 11562.371} C_VEL
LIN {X 0,Y 414.915,Z 823.042,A -85,B 0,C 180,E1 11564.895,E2 11564.895} C_VEL
LIN {X 0,Y 406.125,Z 859.23,A -85,B 0,C 180,E1 11568.196,E2 11568.196} C_VEL
LIN {X 0,Y 396.994,Z 892.805,A -85,B 0,C 180,E1 11572.394,E2 11572.394} C_VEL
LIN {X 0,Y 388.545,Z 921.896,A -85,B 0,C 180,E1 11577.269,E2 11577.269} C_VEL
LIN {X 0,Y 381.545,Z 947.212,A -85,B 0,C 180,E1 11583.014,E2 11583.014} C_VEL
LIN {X 0,Y 376.635,Z 967.596,A -85,B 0,C 180,E1 11589.405,E2 11589.405} C_VEL
LIN {X 0,Y 374.167,Z 981.924,A -85,B 0,C 180,E1 11595.948,E2 11595.948} C_VEL
LIN {X 0,Y 373.243,Z 989.913,A -85,B 0,C 180,E1 11601.837,E2 11601.837} C_VEL
LIN {X 0,Y 373.032,Z 993.712,A -85,B 0,C 180,E1 11607.673,E2 11607.673} C_VEL
LIN {X 0,Y 373.019,Z 993.687,A -85,B 0,C 180,E1 11612.326,E2 11612.326} C_VEL
LIN {X 0,Y 373.229,Z 989.824,A -85,B 0,C 180,E1 11618.162,E2 11618.162} C_VEL
LIN {X 0,Y 374.235,Z 981.755,A -85,B 0,C 180,E1 11624.048,E2 11624.048} C_VEL
LIN {X 0,Y 376.689,Z 967.371,A -85,B 0,C 180,E1 11630.591,E2 11630.591} C_VEL
LIN {X 0,Y 381.593,Z 946.847,A -85,B 0,C 180,E1 11636.996,E2 11636.996} C_VEL
LIN {X 0,Y 388.671,Z 921.492,A -85,B 0,C 180,E1 11642.718,E2 11642.718} C_VEL
LIN {X 0,Y 397.547,Z 890.981,A -85,B 0,C 180,E1 11647.781,E2 11647.781} C_VEL
LIN {X 0,Y 407.056,Z 856.13,A -85,B 0,C 180,E1 11652.03,E2 11652.03} C_VEL
LIN {X 0,Y 416.052,Z 818.109,A -85,B 0,C 180,E1 11655.39,E2 11655.39} C_VEL
LIN {X 0,Y 422.337,Z 783.871,A -85,B 0,C 180,E1 11657.595,E2 11657.595} C_VEL
LIN {X 0,Y 410.385,Z 754.28,A -85,B 0,C 180,E1 11661.722,E2 11661.722} C_VEL
LIN {X 0,Y 395.345,Z 727.262,A -85,B 0,C 180,E1 11666.279,E2 11666.279} C_VEL
LIN {X 0,Y 380.649,Z 705.15,A -85,B 0,C 180,E1 11670.875,E2 11670.875} C_VEL
LIN {X 0,Y 375.521,Z 698.192,A -85,B 0,C 180,E1 11672.614,E2 11672.614} C_VEL
LIN {X 0,Y 372.018,Z 693.55,A -85,B 0,C 180,E1 11673.889,E2 11673.889} C_VEL
LIN {X 0,Y 371.717,Z 691.44,A -85,B 0,C 180,E1 11674.22,E2 11674.22} C_VEL
LIN {X 0,Y 372.003,Z 691.44,A -85,B 0,C 180,E1 11681.006,E2 11681.006} C_VEL
LIN {X 0,Y 372.329,Z 691.44,A -85,B 0,C 180,E1 11688.276,E2 11688.276} C_VEL
LIN {X 0,Y 372.718,Z 691.44,A -85,B 0,C 180,E1 11695.346,E2 11695.346} C_VEL
LIN {X 0,Y 372.887,Z 691.44,A -85,B 0,C 180,E1 11702.332,E2 11702.332} C_VEL
LIN {X 0,Y 372.362,Z 691.44,A -85,B 0,C 180,E1 11709.365,E2 11709.365} C_VEL
LIN {X 0,Y 372.086,Z 691.44,A -85,B 0,C 180,E1 11716.553,E2 11716.553} C_VEL
LIN {X 0,Y 371.725,Z 691.44,A -85,B 0,C 180,E1 11724.039,E2 11724.039} C_VEL
LIN {X 0,Y 371.723,Z 692.088,A -85,B 0,C 180,E1 11725.381,E2 11725.381} C_VEL
LIN {X 0,Y 374.121,Z 697.105,A -85,B 0,C 180,E1 11726.346,E2 11726.346} C_VEL
LIN {X 0,Y 377.018,Z 700.03,A -85,B 0,C 180,E1 11727.329,E2 11727.329} C_VEL
LIN {X 0,Y 394.816,Z 725.334,A -85,B 0,C 180,E1 11732.776,E2 11732.776} C_VEL
LIN {X 0,Y 411.942,Z 754.144,A -85,B 0,C 180,E1 11737.417,E2 11737.417} C_VEL
LIN {X 0,Y 425.116,Z 783.264,A -85,B 0,C 180,E1 11741.216,E2 11741.216} C_VEL
LIN {X 0,Y 417.797,Z 827.021,A -85,B 0,C 180,E1 11743.549,E2 11743.549} C_VEL
LIN {X 0,Y 408.994,Z 866.345,A -85,B 0,C 180,E1 11746.582,E2 11746.582} C_VEL
LIN {X 0,Y 399.38,Z 903.712,A -85,B 0,C 180,E1 11750.623,E2 11750.623} C_VEL
LIN {X 0,Y 390.42,Z 936.44,A -85,B 0,C 180,E1 11755.447,E2 11755.447} C_VEL
LIN {X 0,Y 383.035,Z 964,A -85,B 0,C 180,E1 11760.901,E2 11760.901} C_VEL
LIN {X 0,Y 377.552,Z 987.636,A -85,B 0,C 180,E1 11767.269,E2 11767.269} C_VEL
LIN {X 0,Y 374.602,Z 1004.257,A -85,B 0,C 180,E1 11773.565,E2 11773.565} C_VEL
LIN {X 0,Y 373.369,Z 1015.082,A -85,B 0,C 180,E1 11779.762,E2 11779.762} C_VEL
LIN {X 0,Y 373.033,Z 1020.27,A -85,B 0,C 180,E1 11784.921,E2 11784.921} C_VEL
LIN {X 0,Y 370.648,Z 1021.388,A -85,B 0,C 180,E1 11786.897,E2 11786.897} C_VEL
LIN {X 0,Y 365.181,Z 1021.682,A -85,B 0,C 180,E1 11790.23,E2 11790.23} C_VEL
LIN {X 0,Y 365.133,Z 1019.646,A -85,B 0,C 180,E1 11795.639,E2 11795.639} C_VEL
LIN {X 0,Y 365.681,Z 1012.765,A -85,B 0,C 180,E1 11801.948,E2 11801.948} C_VEL
LIN {X 0,Y 367.518,Z 999.774,A -85,B 0,C 180,E1 11808.646,E2 11808.646} C_VEL
LIN {X 0,Y 371.577,Z 980.462,A -85,B 0,C 180,E1 11815.332,E2 11815.332} C_VEL
LIN {X 0,Y 378.233,Z 955.047,A -85,B 0,C 180,E1 11821.633,E2 11821.633} C_VEL
LIN {X 0,Y 386.96,Z 924.647,A -85,B 0,C 180,E1 11827.143,E2 11827.143} C_VEL
LIN {X 0,Y 396.945,Z 889.333,A -85,B 0,C 180,E1 11831.833,E2 11831.833} C_VEL
LIN {X 0,Y 406.829,Z 850.936,A -85,B 0,C 180,E1 11835.515,E2 11835.515} C_VEL
LIN {X 0,Y 415.386,Z 811.496,A -85,B 0,C 180,E1 11838.178,E2 11838.178} C_VEL
LIN {X 0,Y 419.341,Z 786.342,A -85,B 0,C 180,E1 11839.465,E2 11839.465} C_VEL
LIN {X 0,Y 405.651,Z 755.739,A -85,B 0,C 180,E1 11843.663,E2 11843.663} C_VEL
LIN {X 0,Y 389.229,Z 728.488,A -85,B 0,C 180,E1 11848.405,E2 11848.405} C_VEL
LIN {X 0,Y 377.003,Z 711.001,A -85,B 0,C 180,E1 11852.273,E2 11852.273} C_VEL
LIN {X 0,Y 372.303,Z 704.661,A -85,B 0,C 180,E1 11853.936,E2 11853.936} C_VEL
LIN {X 0,Y 368.108,Z 698.474,A -85,B 0,C 180,E1 11855.571,E2 11855.571} C_VEL
LIN {X 0,Y 364.176,Z 693.894,A -85,B 0,C 180,E1 11857.18,E2 11857.18} C_VEL
LIN {X 0,Y 363.837,Z 691.44,A -85,B 0,C 180,E1 11857.605,E2 11857.605} C_VEL
LIN {X 0,Y 364.07,Z 691.44,A -85,B 0,C 180,E1 11863.072,E2 11863.072} C_VEL
LIN {X 0,Y 364.37,Z 691.44,A -85,B 0,C 180,E1 11870.428,E2 11870.428} C_VEL
LIN {X 0,Y 364.964,Z 691.44,A -85,B 0,C 180,E1 11877.617,E2 11877.617} C_VEL
LIN {X 0,Y 364.703,Z 691.44,A -85,B 0,C 180,E1 11884.877,E2 11884.877} C_VEL
LIN {X 0,Y 364.33,Z 691.44,A -85,B 0,C 180,E1 11891.985,E2 11891.985} C_VEL
LIN {X 0,Y 364.064,Z 691.44,A -85,B 0,C 180,E1 11899.424,E2 11899.424} C_VEL
LIN {X 0,Y 363.835,Z 692.21,A -85,B 0,C 180,E1 11903.093,E2 11903.093} C_VEL
LIN {X 0,Y 366.42,Z 697.289,A -85,B 0,C 180,E1 11904.275,E2 11904.275} C_VEL
LIN {X 0,Y 369.255,Z 699.753,A -85,B 0,C 180,E1 11905.353,E2 11905.353} C_VEL
LIN {X 0,Y 373.318,Z 705.437,A -85,B 0,C 180,E1 11906.892,E2 11906.892} C_VEL
LIN {X 0,Y 388.089,Z 727.25,A -85,B 0,C 180,E1 11911.935,E2 11911.935} C_VEL
LIN {X 0,Y 402.511,Z 752.917,A -85,B 0,C 180,E1 11916.599,E2 11916.599} C_VEL
LIN {X 0,Y 415.011,Z 782.467,A -85,B 0,C 180,E1 11921.034,E2 11921.034} C_VEL
LIN {X 0,Y 416.518,Z 789.537,A -85,B 0,C 180,E1 11921.859,E2 11921.859} C_VEL
LIN {X 0,Y 408.353,Z 827.737,A -85,B 0,C 180,E1 11924.46,E2 11924.46} C_VEL
LIN {X 0,Y 399.006,Z 863.823,A -85,B 0,C 180,E1 11927.909,E2 11927.909} C_VEL
LIN {X 0,Y 389.577,Z 896.287,A -85,B 0,C 180,E1 11932.144,E2 11932.144} C_VEL
LIN {X 0,Y 380.807,Z 925.063,A -85,B 0,C 180,E1 11937.198,E2 11937.198} C_VEL
LIN {X 0,Y 373.692,Z 949.529,A -85,B 0,C 180,E1 11943.018,E2 11943.018} C_VEL
LIN {X 0,Y 369.034,Z 967.898,A -85,B 0,C 180,E1 11948.961,E2 11948.961} C_VEL
LIN {X 0,Y 366.382,Z 982.224,A -85,B 0,C 180,E1 11955.643,E2 11955.643} C_VEL
LIN {X 0,Y 365.386,Z 990.21,A -85,B 0,C 180,E1 11961.66,E2 11961.66} C_VEL
LIN {X 0,Y 365.133,Z 994.008,A -85,B 0,C 180,E1 11967.623,E2 11967.623} C_VEL
LIN {X 0,Y 365.119,Z 993.984,A -85,B 0,C 180,E1 11972.376,E2 11972.376} C_VEL
LIN {X 0,Y 365.374,Z 990.122,A -85,B 0,C 180,E1 11978.339,E2 11978.339} C_VEL
LIN {X 0,Y 366.438,Z 982.058,A -85,B 0,C 180,E1 11984.354,E2 11984.354} C_VEL
LIN {X 0,Y 369.077,Z 967.678,A -85,B 0,C 180,E1 11991.036,E2 11991.036} C_VEL
LIN {X 0,Y 374.371,Z 947.089,A -85,B 0,C 180,E1 11997.58,E2 11997.58} C_VEL
LIN {X 0,Y 381.856,Z 921.8,A -85,B 0,C 180,E1 12003.377,E2 12003.377} C_VEL
LIN {X 0,Y 391.116,Z 891.403,A -85,B 0,C 180,E1 12008.495,E2 12008.495} C_VEL
LIN {X 0,Y 401.113,Z 856.437,A -85,B 0,C 180,E1 12012.8,E2 12012.8} C_VEL
LIN {X 0,Y 410.473,Z 818.428,A -85,B 0,C 180,E1 12016.184,E2 12016.184} C_VEL
LIN {X 0,Y 416.594,Z 787.437,A -85,B 0,C 180,E1 12018.202,E2 12018.202} C_VEL
LIN {X 0,Y 405.141,Z 758.324,A -85,B 0,C 180,E1 12022.419,E2 12022.419} C_VEL
LIN {X 0,Y 389.985,Z 730.345,A -85,B 0,C 180,E1 12027.335,E2 12027.335} C_VEL
LIN {X 0,Y 376.777,Z 710.864,A -85,B 0,C 180,E1 12031.709,E2 12031.709} C_VEL
LIN {X 0,Y 372.241,Z 704.633,A -85,B 0,C 180,E1 12033.342,E2 12033.342} C_VEL
LIN {X 0,Y 367.769,Z 698.279,A -85,B 0,C 180,E1 12035.074,E2 12035.074} C_VEL
LIN {X 0,Y 364.054,Z 693.445,A -85,B 0,C 180,E1 12036.619,E2 12036.619} C_VEL
LIN {X 0,Y 363.795,Z 691.44,A -85,B 0,C 180,E1 12037.006,E2 12037.006} C_VEL
LIN {X 0,Y 364.221,Z 691.44,A -85,B 0,C 180,E1 12043.091,E2 12043.091} C_VEL
LIN {X 0,Y 364.488,Z 691.44,A -85,B 0,C 180,E1 12050.443,E2 12050.443} C_VEL
LIN {X 0,Y 364.93,Z 691.44,A -85,B 0,C 180,E1 12057.628,E2 12057.628} C_VEL
LIN {X 0,Y 364.97,Z 691.44,A -85,B 0,C 180,E1 12062.383,E2 12062.383} C_VEL
LIN {X 0,Y 364.421,Z 691.44,A -85,B 0,C 180,E1 12069.571,E2 12069.571} C_VEL
LIN {X 0,Y 364.125,Z 691.44,A -85,B 0,C 180,E1 12076.988,E2 12076.988} C_VEL
LIN {X 0,Y 363.818,Z 691.93,A -85,B 0,C 180,E1 12082.646,E2 12082.646} C_VEL
LIN {X 0,Y 366.037,Z 696.951,A -85,B 0,C 180,E1 12083.692,E2 12083.692} C_VEL
LIN {X 0,Y 369.349,Z 700.166,A -85,B 0,C 180,E1 12084.967,E2 12084.967} C_VEL
LIN {X 0,Y 380.207,Z 715.442,A -85,B 0,C 180,E1 12088.826,E2 12088.826} C_VEL
LIN {X 0,Y 394.989,Z 737.2,A -85,B 0,C 180,E1 12093.274,E2 12093.274} C_VEL
LIN {X 0,Y 409.884,Z 764.424,A -85,B 0,C 180,E1 12097.608,E2 12097.608} C_VEL
LIN {X 0,Y 419.435,Z 786.761,A -85,B 0,C 180,E1 12100.587,E2 12100.587} C_VEL
LIN {X 0,Y 412.276,Z 826.713,A -85,B 0,C 180,E1 12102.736,E2 12102.736} C_VEL
LIN {X 0,Y 403.193,Z 865.74,A -85,B 0,C 180,E1 12105.76,E2 12105.76} C_VEL
LIN {X 0,Y 392.974,Z 903.613,A -85,B 0,C 180,E1 12109.888,E2 12109.888} C_VEL
LIN {X 0,Y 383.575,Z 936.125,A -85,B 0,C 180,E1 12114.74,E2 12114.74} C_VEL
LIN {X 0,Y 375.747,Z 964.049,A -85,B 0,C 180,E1 12120.373,E2 12120.373} C_VEL
LIN {X 0,Y 370.002,Z 987.328,A -85,B 0,C 180,E1 12126.779,E2 12126.779} C_VEL
LIN {X 0,Y 366.828,Z 1003.953,A -85,B 0,C 180,E1 12133.207,E2 12133.207} C_VEL
LIN {X 0,Y 365.544,Z 1014.407,A -85,B 0,C 180,E1 12139.258,E2 12139.258} C_VEL
LIN {X 0,Y 365.156,Z 1020.294,A -85,B 0,C 180,E1 12145.244,E2 12145.244} C_VEL
LIN {X 0,Y 365.181,Z 1021.682,A -85,B 0,C 180,E1 12150.23,E2 12150.23} C_VEL
LIN {X 0,Y 361.106,Z 1020.995,A -85,B 0,C 180,E1 12152.906,E2 12152.906} C_VEL
LIN {X 0,Y 357.22,Z 1019.436,A -85,B 0,C 180,E1 12155.632,E2 12155.632} C_VEL
LIN {X 0,Y 357.679,Z 1014.105,A -85,B 0,C 180,E1 12160.982,E2 12160.982} C_VEL
LIN {X 0,Y 359.059,Z 1003.648,A -85,B 0,C 180,E1 12167.169,E2 12167.169} C_VEL
LIN {X 0,Y 362.384,Z 987.215,A -85,B 0,C 180,E1 12173.666,E2 12173.666} C_VEL
LIN {X 0,Y 368.264,Z 964.702,A -85,B 0,C 180,E1 12180.026,E2 12180.026} C_VEL
LIN {X 0,Y 376.957,Z 935.866,A -85,B 0,C 180,E1 12185.967,E2 12185.967} C_VEL
LIN {X 0,Y 386.969,Z 902.775,A -85,B 0,C 180,E1 12190.963,E2 12190.963} C_VEL
LIN {X 0,Y 397.406,Z 865.694,A -85,B 0,C 180,E1 12195.033,E2 12195.033} C_VEL
LIN {X 0,Y 406.878,Z 826.477,A -85,B 0,C 180,E1 12198.095,E2 12198.095} C_VEL
LIN {X 0,Y 413.558,Z 789.527,A -85,B 0,C 180,E1 12200.158,E2 12200.158} C_VEL
LIN {X 0,Y 400.215,Z 759.154,A -85,B 0,C 180,E1 12204.515,E2 12204.515} C_VEL
LIN {X 0,Y 383.747,Z 731.133,A -85,B 0,C 180,E1 12209.632,E2 12209.632} C_VEL
LIN {X 0,Y 370.405,Z 712.139,A -85,B 0,C 180,E1 12214.211,E2 12214.211} C_VEL
LIN {X 0,Y 365.083,Z 705.164,A -85,B 0,C 180,E1 12216.306,E2 12216.306} C_VEL
LIN {X 0,Y 361.369,Z 699.341,A -85,B 0,C 180,E1 12217.967,E2 12217.967} C_VEL
LIN {X 0,Y 356.706,Z 694.557,A -85,B 0,C 180,E1 12220.146,E2 12220.146} C_VEL
LIN {X 0,Y 356.086,Z 691.44,A -85,B 0,C 180,E1 12220.756,E2 12220.756} C_VEL
LIN {X 0,Y 356.287,Z 691.44,A -85,B 0,C 180,E1 12227.801,E2 12227.801} C_VEL
LIN {X 0,Y 356.792,Z 691.44,A -85,B 0,C 180,E1 12235.126,E2 12235.126} C_VEL
LIN {X 0,Y 357.1,Z 691.44,A -85,B 0,C 180,E1 12239.994,E2 12239.994} C_VEL
LIN {X 0,Y 356.657,Z 691.44,A -85,B 0,C 180,E1 12247.31,E2 12247.31} C_VEL
LIN {X 0,Y 356.27,Z 691.44,A -85,B 0,C 180,E1 12254.765,E2 12254.765} C_VEL
LIN {X 0,Y 356.077,Z 691.478,A -85,B 0,C 180,E1 12259.878,E2 12259.878} C_VEL
LIN {X 0,Y 357.679,Z 696.337,A -85,B 0,C 180,E1 12260.858,E2 12260.858} C_VEL
LIN {X 0,Y 361.693,Z 700.325,A -85,B 0,C 180,E1 12262.691,E2 12262.691} C_VEL
LIN {X 0,Y 366.377,Z 706.025,A -85,B 0,C 180,E1 12264.668,E2 12264.668} C_VEL
LIN {X 0,Y 380.816,Z 727.486,A -85,B 0,C 180,E1 12270.118,E2 12270.118} C_VEL
LIN {X 0,Y 394.141,Z 750.495,A -85,B 0,C 180,E1 12274.709,E2 12274.709} C_VEL
LIN {X 0,Y 406.588,Z 778.518,A -85,B 0,C 180,E1 12279.263,E2 12279.263} C_VEL
LIN {X 0,Y 410.75,Z 792.491,A -85,B 0,C 180,E1 12281.187,E2 12281.187} C_VEL
LIN {X 0,Y 402.052,Z 831.391,A -85,B 0,C 180,E1 12283.926,E2 12283.926} C_VEL
LIN {X 0,Y 391.703,Z 869.01,A -85,B 0,C 180,E1 12287.676,E2 12287.676} C_VEL
LIN {X 0,Y 381.183,Z 903.077,A -85,B 0,C 180,E1 12292.414,E2 12292.414} C_VEL
LIN {X 0,Y 371.796,Z 932.401,A -85,B 0,C 180,E1 12298.034,E2 12298.034} C_VEL
LIN {X 0,Y 364.731,Z 955.689,A -85,B 0,C 180,E1 12304.158,E2 12304.158} C_VEL
LIN {X 0,Y 360.216,Z 973.935,A -85,B 0,C 180,E1 12310.91,E2 12310.91} C_VEL
LIN {X 0,Y 357.974,Z 986.294,A -85,B 0,C 180,E1 12317.79,E2 12317.79} C_VEL
LIN {X 0,Y 357.424,Z 991.668,A -85,B 0,C 180,E1 12322.698,E2 12322.698} C_VEL
LIN {X 0,Y 357.246,Z 994.304,A -85,B 0,C 180,E1 12327.57,E2 12327.57} C_VEL
LIN {X 0,Y 357.231,Z 994.281,A -85,B 0,C 180,E1 12332.429,E2 12332.429} C_VEL
LIN {X 0,Y 357.514,Z 990.421,A -85,B 0,C 180,E1 12338.524,E2 12338.524} C_VEL
LIN {X 0,Y 358.644,Z 982.362,A -85,B 0,C 180,E1 12344.672,E2 12344.672} C_VEL
LIN {X 0,Y 361.493,Z 967.986,A -85,B 0,C 180,E1 12351.499,E2 12351.499} C_VEL
LIN {X 0,Y 366.9,Z 948.245,A -85,B 0,C 180,E1 12357.932,E2 12357.932} C_VEL
LIN {X 0,Y 375.003,Z 922.309,A -85,B 0,C 180,E1 12364.022,E2 12364.022} C_VEL
LIN {X 0,Y 385.024,Z 890.884,A -85,B 0,C 180,E1 12369.367,E2 12369.367} C_VEL
LIN {X 0,Y 395.249,Z 856.744,A -85,B 0,C 180,E1 12373.592,E2 12373.592} C_VEL
LIN {X 0,Y 405.008,Z 818.721,A -85,B 0,C 180,E1 12376.997,E2 12376.997} C_VEL
LIN {X 0,Y 410.917,Z 791.059,A -85,B 0,C 180,E1 12378.818,E2 12378.818} C_VEL
LIN {X 0,Y 399.491,Z 761.544,A -85,B 0,C 180,E1 12383.284,E2 12383.284} C_VEL
LIN {X 0,Y 385.666,Z 735.411,A -85,B 0,C 180,E1 12388.089,E2 12388.089} C_VEL
LIN {X 0,Y 373.654,Z 717.139,A -85,B 0,C 180,E1 12392.318,E2 12392.318} C_VEL
LIN {X 0,Y 365.264,Z 705.282,A -85,B 0,C 180,E1 12395.613,E2 12395.613} C_VEL
LIN {X 0,Y 361.445,Z 699.591,A -85,B 0,C 180,E1 12397.293,E2 12397.293} C_VEL
LIN {X 0,Y 356.44,Z 693.987,A -85,B 0,C 180,E1 12399.651,E2 12399.651} C_VEL
LIN {X 0,Y 356.084,Z 691.44,A -85,B 0,C 180,E1 12400.122,E2 12400.122} C_VEL
LIN {X 0,Y 356.461,Z 691.44,A -85,B 0,C 180,E1 12407.746,E2 12407.746} C_VEL
LIN {X 0,Y 356.909,Z 691.44,A -85,B 0,C 180,E1 12415.14,E2 12415.14} C_VEL
LIN {X 0,Y 357.081,Z 691.44,A -85,B 0,C 180,E1 12422.436,E2 12422.436} C_VEL
LIN {X 0,Y 356.481,Z 691.44,A -85,B 0,C 180,E1 12429.786,E2 12429.786} C_VEL
LIN {X 0,Y 356.198,Z 691.44,A -85,B 0,C 180,E1 12437.314,E2 12437.314} C_VEL
LIN {X 0,Y 356.112,Z 691.466,A -85,B 0,C 180,E1 12439.484,E2 12439.484} C_VEL
LIN {X 0,Y 357.75,Z 696.439,A -85,B 0,C 180,E1 12440.48,E2 12440.48} C_VEL
LIN {X 0,Y 361.634,Z 700.224,A -85,B 0,C 180,E1 12442.239,E2 12442.239} C_VEL
LIN {X 0,Y 366.075,Z 705.854,A -85,B 0,C 180,E1 12444.123,E2 12444.123} C_VEL
LIN {X 0,Y 381.056,Z 727.208,A -85,B 0,C 180,E1 12449.536,E2 12449.536} C_VEL
LIN {X 0,Y 396.333,Z 752.067,A -85,B 0,C 180,E1 12454.298,E2 12454.298} C_VEL
LIN {X 0,Y 410.072,Z 780.543,A -85,B 0,C 180,E1 12458.64,E2 12458.64} C_VEL
LIN {X 0,Y 413.633,Z 790.706,A -85,B 0,C 180,E1 12459.949,E2 12459.949} C_VEL
LIN {X 0,Y 406.148,Z 829.465,A -85,B 0,C 180,E1 12462.11,E2 12462.11} C_VEL
LIN {X 0,Y 396.801,Z 867.59,A -85,B 0,C 180,E1 12465.147,E2 12465.147} C_VEL
LIN {X 0,Y 386.481,Z 904.088,A -85,B 0,C 180,E1 12469.209,E2 12469.209} C_VEL
LIN {X 0,Y 376.836,Z 935.919,A -85,B 0,C 180,E1 12474.036,E2 12474.036} C_VEL
LIN {X 0,Y 368.305,Z 964.649,A -85,B 0,C 180,E1 12479.965,E2 12479.965} C_VEL
LIN {X 0,Y 362.462,Z 986.961,A -85,B 0,C 180,E1 12486.245,E2 12486.245} C_VEL
LIN {X 0,Y 359.072,Z 1003.649,A -85,B 0,C 180,E1 12492.833,E2 12492.833} C_VEL
LIN {X 0,Y 357.658,Z 1014.106,A -85,B 0,C 180,E1 12499.019,E2 12499.019} C_VEL
LIN {X 0,Y 357.261,Z 1019.997,A -85,B 0,C 180,E1 12505.138,E2 12505.138} C_VEL
LIN {X 0,Y 357.291,Z 1021.391,A -85,B 0,C 180,E1 12510.199,E2 12510.199} C_VEL
LIN {X 0,Y 357.22,Z 1019.436,A -85,B 0,C 180,E1 12515.632,E2 12515.632} C_VEL
LIN {X 0,Y 354.778,Z 1017.788,A -85,B 0,C 180,E1 12517.692,E2 12517.692} C_VEL
LIN {X 0,Y 349.819,Z 1014.386,A -85,B 0,C 180,E1 12520.78,E2 12520.78} C_VEL
LIN {X 0,Y 349.784,Z 1013.931,A -85,B 0,C 180,E1 12521.134,E2 12521.134} C_VEL
LIN {X 0,Y 351.296,Z 1003.343,A -85,B 0,C 180,E1 12527.56,E2 12527.56} C_VEL
LIN {X 0,Y 354.993,Z 986.386,A -85,B 0,C 180,E1 12534.382,E2 12534.382} C_VEL
LIN {X 0,Y 361.701,Z 962.664,A -85,B 0,C 180,E1 12541.105,E2 12541.105} C_VEL
LIN {X 0,Y 370.527,Z 934.722,A -85,B 0,C 180,E1 12546.873,E2 12546.873} C_VEL
LIN {X 0,Y 381.17,Z 901.281,A -85,B 0,C 180,E1 12551.923,E2 12551.923} C_VEL
LIN {X 0,Y 391.835,Z 864.814,A -85,B 0,C 180,E1 12555.93,E2 12555.93} C_VEL
LIN {X 0,Y 401.832,Z 825.054,A -85,B 0,C 180,E1 12559.02,E2 12559.02} C_VEL
LIN {X 0,Y 407.833,Z 792.761,A -85,B 0,C 180,E1 12560.867,E2 12560.867} C_VEL
LIN {X 0,Y 395.236,Z 763.469,A -85,B 0,C 180,E1 12565.26,E2 12565.26} C_VEL
LIN {X 0,Y 380.297,Z 737.213,A -85,B 0,C 180,E1 12570.235,E2 12570.235} C_VEL
LIN {X 0,Y 367.731,Z 718.798,A -85,B 0,C 180,E1 12574.78,E2 12574.78} C_VEL
LIN {X 0,Y 362.481,Z 711.932,A -85,B 0,C 180,E1 12576.916,E2 12576.916} C_VEL
LIN {X 0,Y 357.976,Z 705.684,A -85,B 0,C 180,E1 12578.986,E2 12578.986} C_VEL
LIN {X 0,Y 354.141,Z 700.196,A -85,B 0,C 180,E1 12580.97,E2 12580.97} C_VEL
LIN {X 0,Y 351.679,Z 697.998,A -85,B 0,C 180,E1 12582.295,E2 12582.295} C_VEL
LIN {X 0,Y 348.357,Z 693.173,A -85,B 0,C 180,E1 12584.42,E2 12584.42} C_VEL
LIN {X 0,Y 348.19,Z 691.44,A -85,B 0,C 180,E1 12584.872,E2 12584.872} C_VEL
LIN {X 0,Y 348.717,Z 691.44,A -85,B 0,C 180,E1 12592.511,E2 12592.511} C_VEL
LIN {X 0,Y 349.198,Z 691.44,A -85,B 0,C 180,E1 12599.994,E2 12599.994} C_VEL
LIN {X 0,Y 348.734,Z 691.44,A -85,B 0,C 180,E1 12607.477,E2 12607.477} C_VEL
LIN {X 0,Y 348.324,Z 691.44,A -85,B 0,C 180,E1 12615.11,E2 12615.11} C_VEL
LIN {X 0,Y 348.321,Z 692.201,A -85,B 0,C 180,E1 12615.97,E2 12615.97} C_VEL
LIN {X 0,Y 350.753,Z 697.173,A -85,B 0,C 180,E1 12617.66,E2 12617.66} C_VEL
LIN {X 0,Y 354.014,Z 699.797,A -85,B 0,C 180,E1 12619.429,E2 12619.429} C_VEL
LIN {X 0,Y 357.735,Z 705.491,A -85,B 0,C 180,E1 12621.387,E2 12621.387} C_VEL
LIN {X 0,Y 359.896,Z 708.244,A -85,B 0,C 180,E1 12622.402,E2 12622.402} C_VEL
LIN {X 0,Y 366.1,Z 716.988,A -85,B 0,C 180,E1 12625.153,E2 12625.153} C_VEL
LIN {X 0,Y 376.934,Z 732.674,A -85,B 0,C 180,E1 12629.383,E2 12629.383} C_VEL
LIN {X 0,Y 390.542,Z 757.532,A -85,B 0,C 180,E1 12634.459,E2 12634.459} C_VEL
LIN {X 0,Y 402.209,Z 785.538,A -85,B 0,C 180,E1 12639.103,E2 12639.103} C_VEL
LIN {X 0,Y 405.055,Z 795.103,A -85,B 0,C 180,E1 12640.483,E2 12640.483} C_VEL
LIN {X 0,Y 396.494,Z 831.799,A -85,B 0,C 180,E1 12643.1,E2 12643.1} C_VEL
LIN {X 0,Y 385.967,Z 868.723,A -85,B 0,C 180,E1 12646.803,E2 12646.803} C_VEL
LIN {X 0,Y 374.873,Z 903.171,A -85,B 0,C 180,E1 12651.624,E2 12651.624} C_VEL
LIN {X 0,Y 364.925,Z 932.704,A -85,B 0,C 180,E1 12657.358,E2 12657.358} C_VEL
LIN {X 0,Y 357.311,Z 956.153,A -85,B 0,C 180,E1 12663.637,E2 12663.637} C_VEL
LIN {X 0,Y 352.541,Z 974.347,A -85,B 0,C 180,E1 12670.533,E2 12670.533} C_VEL
LIN {X 0,Y 350.151,Z 986.593,A -85,B 0,C 180,E1 12677.513,E2 12677.513} C_VEL
LIN {X 0,Y 349.558,Z 991.964,A -85,B 0,C 180,E1 12682.533,E2 12682.533} C_VEL
LIN {X 0,Y 349.347,Z 994.601,A -85,B 0,C 180,E1 12687.516,E2 12687.516} C_VEL
LIN {X 0,Y 349.33,Z 994.577,A -85,B 0,C 180,E1 12692.484,E2 12692.484} C_VEL
LIN {X 0,Y 349.641,Z 990.721,A -85,B 0,C 180,E1 12698.717,E2 12698.717} C_VEL
LIN {X 0,Y 350.857,Z 982.665,A -85,B 0,C 180,E1 12705.006,E2 12705.006} C_VEL
LIN {X 0,Y 353.935,Z 968.292,A -85,B 0,C 180,E1 12711.981,E2 12711.981} C_VEL
LIN {X 0,Y 360.116,Z 947.216,A -85,B 0,C 180,E1 12718.914,E2 12718.914} C_VEL
LIN {X 0,Y 368.87,Z 920.857,A -85,B 0,C 180,E1 12725.075,E2 12725.075} C_VEL
LIN {X 0,Y 378.714,Z 891.474,A -85,B 0,C 180,E1 12730.104,E2 12730.104} C_VEL
LIN {X 0,Y 389.456,Z 857.051,A -85,B 0,C 180,E1 12734.409,E2 12734.409} C_VEL
LIN {X 0,Y 399.605,Z 819.027,A -85,B 0,C 180,E1 12737.834,E2 12737.834} C_VEL
LIN {X 0,Y 404.986,Z 793.938,A -85,B 0,C 180,E1 12739.542,E2 12739.542} C_VEL
LIN {X 0,Y 394.185,Z 765.35,A -85,B 0,C 180,E1 12744.068,E2 12744.068} C_VEL
LIN {X 0,Y 380.093,Z 737.948,A -85,B 0,C 180,E1 12749.322,E2 12749.322} C_VEL
LIN {X 0,Y 367.177,Z 718.464,A -85,B 0,C 180,E1 12754.272,E2 12754.272} C_VEL
LIN {X 0,Y 362.22,Z 711.733,A -85,B 0,C 180,E1 12756.367,E2 12756.367} C_VEL
LIN {X 0,Y 357.942,Z 705.64,A -85,B 0,C 180,E1 12758.365,E2 12758.365} C_VEL
LIN {X 0,Y 354.11,Z 700.243,A -85,B 0,C 180,E1 12760.332,E2 12760.332} C_VEL
LIN {X 0,Y 352.192,Z 698.317,A -85,B 0,C 180,E1 12761.362,E2 12761.362} C_VEL
LIN {X 0,Y 348.527,Z 693.177,A -85,B 0,C 180,E1 12763.645,E2 12763.645} C_VEL
LIN {X 0,Y 348.334,Z 691.44,A -85,B 0,C 180,E1 12764.019,E2 12764.019} C_VEL
LIN {X 0,Y 348.614,Z 691.44,A -85,B 0,C 180,E1 12771.247,E2 12771.247} C_VEL
LIN {X 0,Y 349.136,Z 691.44,A -85,B 0,C 180,E1 12777.521,E2 12777.521} C_VEL
LIN {X 0,Y 348.97,Z 691.44,A -85,B 0,C 180,E1 12783.716,E2 12783.716} C_VEL
LIN {X 0,Y 348.548,Z 691.44,A -85,B 0,C 180,E1 12790.011,E2 12790.011} C_VEL
LIN {X 0,Y 348.284,Z 691.864,A -85,B 0,C 180,E1 12795.546,E2 12795.546} C_VEL
LIN {X 0,Y 350.122,Z 696.526,A -85,B 0,C 180,E1 12796.894,E2 12796.894} C_VEL
LIN {X 0,Y 354.152,Z 700.173,A -85,B 0,C 180,E1 12799.11,E2 12799.11} C_VEL
LIN {X 0,Y 357.979,Z 705.673,A -85,B 0,C 180,E1 12801.08,E2 12801.08} C_VEL
LIN {X 0,Y 360.694,Z 709.74,A -85,B 0,C 180,E1 12802.363,E2 12802.363} C_VEL
LIN {X 0,Y 365.495,Z 715.82,A -85,B 0,C 180,E1 12804.386,E2 12804.386} C_VEL
LIN {X 0,Y 374.652,Z 728.807,A -85,B 0,C 180,E1 12807.86,E2 12807.86} C_VEL
LIN {X 0,Y 388.192,Z 750.351,A -85,B 0,C 180,E1 12812.433,E2 12812.433} C_VEL
LIN {X 0,Y 401.727,Z 777.42,A -85,B 0,C 180,E1 12816.951,E2 12816.951} C_VEL
LIN {X 0,Y 407.883,Z 794.301,A -85,B 0,C 180,E1 12819.267,E2 12819.267} C_VEL
LIN {X 0,Y 399.67,Z 833.808,A -85,B 0,C 180,E1 12821.571,E2 12821.571} C_VEL
LIN {X 0,Y 390.408,Z 869.61,A -85,B 0,C 180,E1 12824.535,E2 12824.535} C_VEL
LIN {X 0,Y 380.104,Z 904.359,A -85,B 0,C 180,E1 12828.479,E2 12828.479} C_VEL
LIN {X 0,Y 369.959,Z 936.272,A -85,B 0,C 180,E1 12833.408,E2 12833.408} C_VEL
LIN {X 0,Y 361.204,Z 964.339,A -85,B 0,C 180,E1 12839.311,E2 12839.311} C_VEL
LIN {X 0,Y 355.02,Z 986.387,A -85,B 0,C 180,E1 12845.619,E2 12845.619} C_VEL
LIN {X 0,Y 351.324,Z 1003.344,A -85,B 0,C 180,E1 12852.442,E2 12852.442} C_VEL
LIN {X 0,Y 349.785,Z 1013.805,A -85,B 0,C 180,E1 12858.768,E2 12858.768} C_VEL
LIN {X 0,Y 349.376,Z 1019.7,A -85,B 0,C 180,E1 12865.028,E2 12865.028} C_VEL
LIN {X 0,Y 349.426,Z 1021.125,A -85,B 0,C 180,E1 12870,E2 12870} C_VEL
LIN {X 0,Y 349.341,Z 1019.235,A -85,B 0,C 180,E1 12875.625,E2 12875.625} C_VEL
LIN {X 0,Y 349.784,Z 1013.931,A -85,B 0,C 180,E1 12881.134,E2 12881.134} C_VEL
LIN {X 0,Y 347.638,Z 1011.124,A -85,B 0,C 180,E1 12883.209,E2 12883.209} C_VEL
LIN {X 0,Y 343.106,Z 1006.133,A -85,B 0,C 180,E1 12886.313,E2 12886.313} C_VEL
LIN {X 0,Y 343.13,Z 1005.488,A -85,B 0,C 180,E1 12886.666,E2 12886.666} C_VEL
LIN {X 0,Y 346.408,Z 990.346,A -85,B 0,C 180,E1 12893.386,E2 12893.386} C_VEL
LIN {X 0,Y 352.327,Z 969.437,A -85,B 0,C 180,E1 12899.972,E2 12899.972} C_VEL
LIN {X 0,Y 360.943,Z 943.346,A -85,B 0,C 180,E1 12905.964,E2 12905.964} C_VEL
LIN {X 0,Y 371.185,Z 912.688,A -85,B 0,C 180,E1 12911.166,E2 12911.166} C_VEL
LIN {X 0,Y 382.662,Z 876.569,A -85,B 0,C 180,E1 12915.61,E2 12915.61} C_VEL
LIN {X 0,Y 393.123,Z 838.645,A -85,B 0,C 180,E1 12918.959,E2 12918.959} C_VEL
LIN {X 0,Y 402.252,Z 796.289,A -85,B 0,C 180,E1 12921.56,E2 12921.56} C_VEL
LIN {X 0,Y 390.257,Z 767.667,A -85,B 0,C 180,E1 12926.034,E2 12926.034} C_VEL
LIN {X 0,Y 376.156,Z 742.3,A -85,B 0,C 180,E1 12931.033,E2 12931.033} C_VEL
LIN {X 0,Y 364.685,Z 725.087,A -85,B 0,C 180,E1 12935.467,E2 12935.467} C_VEL
LIN {X 0,Y 359.83,Z 718.487,A -85,B 0,C 180,E1 12937.581,E2 12937.581} C_VEL
LIN {X 0,Y 355.684,Z 712.721,A -85,B 0,C 180,E1 12939.558,E2 12939.558} C_VEL
LIN {X 0,Y 350.886,Z 706.031,A -85,B 0,C 180,E1 12942.172,E2 12942.172} C_VEL
LIN {X 0,Y 346.725,Z 700.826,A -85,B 0,C 180,E1 12944.807,E2 12944.807} C_VEL
LIN {X 0,Y 345.49,Z 698.872,A -85,B 0,C 180,E1 12945.725,E2 12945.725} C_VEL
LIN {X 0,Y 341.007,Z 694.211,A -85,B 0,C 180,E1 12949.5,E2 12949.5} C_VEL
LIN {X 0,Y 340.588,Z 691.44,A -85,B 0,C 180,E1 12950.399,E2 12950.399} C_VEL
LIN {X 0,Y 341.248,Z 691.44,A -85,B 0,C 180,E1 12957.451,E2 12957.451} C_VEL
LIN {X 0,Y 341.167,Z 691.44,A -85,B 0,C 180,E1 12962.537,E2 12962.537} C_VEL
LIN {X 0,Y 340.635,Z 691.887,A -85,B 0,C 180,E1 12970.379,E2 12970.379} C_VEL
LIN {X 0,Y 342.4,Z 696.496,A -85,B 0,C 180,E1 12972.375,E2 12972.375} C_VEL
LIN {X 0,Y 346.624,Z 700.148,A -85,B 0,C 180,E1 12975.563,E2 12975.563} C_VEL
LIN {X 0,Y 350.46,Z 705.738,A -85,B 0,C 180,E1 12978.077,E2 12978.077} C_VEL
LIN {X 0,Y 352.434,Z 708.095,A -85,B 0,C 180,E1 12979.194,E2 12979.194} C_VEL
LIN {X 0,Y 358.307,Z 716.51,A -85,B 0,C 180,E1 12982.281,E2 12982.281} C_VEL
LIN {X 0,Y 366.64,Z 728.096,A -85,B 0,C 180,E1 12986.015,E2 12986.015} C_VEL
LIN {X 0,Y 380.055,Z 750.546,A -85,B 0,C 180,E1 12991.445,E2 12991.445} C_VEL
LIN {X 0,Y 392.251,Z 777.096,A -85,B 0,C 180,E1 12996.425,E2 12996.425} C_VEL
LIN {X 0,Y 399.212,Z 798.712,A -85,B 0,C 180,E1 12999.823,E2 12999.823} C_VEL
LIN {X 0,Y 390.233,Z 835.065,A -85,B 0,C 180,E1 13002.507,E2 13002.507} C_VEL
LIN {X 0,Y 379.572,Z 870.705,A -85,B 0,C 180,E1 13006.175,E2 13006.175} C_VEL
LIN {X 0,Y 368.301,Z 904.088,A -85,B 0,C 180,E1 13010.945,E2 13010.945} C_VEL
LIN {X 0,Y 358.025,Z 933.009,A -85,B 0,C 180,E1 13016.648,E2 13016.648} C_VEL
LIN {X 0,Y 349.948,Z 956.768,A -85,B 0,C 180,E1 13023.152,E2 13023.152} C_VEL
LIN {X 0,Y 344.98,Z 974.44,A -85,B 0,C 180,E1 13029.981,E2 13029.981} C_VEL
LIN {X 0,Y 342.339,Z 986.892,A -85,B 0,C 180,E1 13037.224,E2 13037.224} C_VEL
LIN {X 0,Y 341.675,Z 992.262,A -85,B 0,C 180,E1 13042.36,E2 13042.36} C_VEL
LIN {X 0,Y 341.462,Z 994.896,A -85,B 0,C 180,E1 13047.458,E2 13047.458} C_VEL
LIN {X 0,Y 341.444,Z 994.874,A -85,B 0,C 180,E1 13052.541,E2 13052.541} C_VEL
LIN {X 0,Y 341.773,Z 991.02,A -85,B 0,C 180,E1 13058.919,E2 13058.919} C_VEL
LIN {X 0,Y 343.078,Z 982.969,A -85,B 0,C 180,E1 13065.354,E2 13065.354} C_VEL
LIN {X 0,Y 346.428,Z 968.598,A -85,B 0,C 180,E1 13072.483,E2 13072.483} C_VEL
LIN {X 0,Y 353.004,Z 947.524,A -85,B 0,C 180,E1 13079.554,E2 13079.554} C_VEL
LIN {X 0,Y 362.237,Z 921.166,A -85,B 0,C 180,E1 13085.815,E2 13085.815} C_VEL
LIN {X 0,Y 372.842,Z 890.816,A -85,B 0,C 180,E1 13091.048,E2 13091.048} C_VEL
LIN {X 0,Y 384.058,Z 856.293,A -85,B 0,C 180,E1 13095.359,E2 13095.359} C_VEL
LIN {X 0,Y 394.29,Z 819.333,A -85,B 0,C 180,E1 13098.694,E2 13098.694} C_VEL
LIN {X 0,Y 399.158,Z 797.273,A -85,B 0,C 180,E1 13100.229,E2 13100.229} C_VEL
LIN {X 0,Y 388.951,Z 769.246,A -85,B 0,C 180,E1 13104.832,E2 13104.832} C_VEL
LIN {X 0,Y 376.08,Z 743.698,A -85,B 0,C 180,E1 13109.963,E2 13109.963} C_VEL
LIN {X 0,Y 364.409,Z 725.095,A -85,B 0,C 180,E1 13114.804,E2 13114.804} C_VEL
LIN {X 0,Y 355.838,Z 712.884,A -85,B 0,C 180,E1 13118.806,E2 13118.806} C_VEL
LIN {X 0,Y 350.99,Z 706.093,A -85,B 0,C 180,E1 13121.459,E2 13121.459} C_VEL
LIN {X 0,Y 346.808,Z 700.621,A -85,B 0,C 180,E1 13124.092,E2 13124.092} C_VEL
LIN {X 0,Y 345.426,Z 698.732,A -85,B 0,C 180,E1 13125.086,E2 13125.086} C_VEL
LIN {X 0,Y 341.011,Z 693.956,A -85,B 0,C 180,E1 13128.775,E2 13128.775} C_VEL
LIN {X 0,Y 340.674,Z 691.44,A -85,B 0,C 180,E1 13129.567,E2 13129.567} C_VEL
LIN {X 0,Y 341.233,Z 691.44,A -85,B 0,C 180,E1 13137.463,E2 13137.463} C_VEL
LIN {X 0,Y 341.254,Z 691.44,A -85,B 0,C 180,E1 13142.549,E2 13142.549} C_VEL
LIN {X 0,Y 340.652,Z 691.744,A -85,B 0,C 180,E1 13150.084,E2 13150.084} C_VEL
LIN {X 0,Y 342.157,Z 696.261,A -85,B 0,C 180,E1 13151.832,E2 13151.832} C_VEL
LIN {X 0,Y 346.626,Z 700.231,A -85,B 0,C 180,E1 13155.198,E2 13155.198} C_VEL
LIN {X 0,Y 350.336,Z 705.657,A -85,B 0,C 180,E1 13157.613,E2 13157.613} C_VEL
LIN {X 0,Y 352.334,Z 707.784,A -85,B 0,C 180,E1 13158.724,E2 13158.724} C_VEL
LIN {X 0,Y 356.758,Z 713.481,A -85,B 0,C 180,E1 13161.001,E2 13161.001} C_VEL
LIN {X 0,Y 368.552,Z 730.614,A -85,B 0,C 180,E1 13166.128,E2 13166.128} C_VEL
LIN {X 0,Y 381.871,Z 751.853,A -85,B 0,C 180,E1 13171.028,E2 13171.028} C_VEL
LIN {X 0,Y 395.348,Z 778.664,A -85,B 0,C 180,E1 13175.821,E2 13175.821} C_VEL
LIN {X 0,Y 402.329,Z 796.669,A -85,B 0,C 180,E1 13178.497,E2 13178.497} C_VEL
LIN {X 0,Y 393.199,Z 838.391,A -85,B 0,C 180,E1 13181.036,E2 13181.036} C_VEL
LIN {X 0,Y 382.27,Z 877.836,A -85,B 0,C 180,E1 13184.526,E2 13184.526} C_VEL
LIN {X 0,Y 370.839,Z 913.768,A -85,B 0,C 180,E1 13188.999,E2 13188.999} C_VEL
LIN {X 0,Y 360.344,Z 944.942,A -85,B 0,C 180,E1 13194.343,E2 13194.343} C_VEL
LIN {X 0,Y 351.579,Z 971.828,A -85,B 0,C 180,E1 13200.669,E2 13200.669} C_VEL
LIN {X 0,Y 345.768,Z 992.684,A -85,B 0,C 180,E1 13207.471,E2 13207.471} C_VEL
LIN {X 0,Y 342.723,Z 1007.845,A -85,B 0,C 180,E1 13214.629,E2 13214.629} C_VEL
LIN {X 0,Y 341.695,Z 1016.382,A -85,B 0,C 180,E1 13221.079,E2 13221.079} C_VEL
LIN {X 0,Y 341.498,Z 1020.472,A -85,B 0,C 180,E1 13227.459,E2 13227.459} C_VEL
LIN {X 0,Y 341.437,Z 1020.469,A -85,B 0,C 180,E1 13232.542,E2 13232.542} C_VEL
LIN {X 0,Y 341.706,Z 1016.382,A -85,B 0,C 180,E1 13238.922,E2 13238.922} C_VEL
LIN {X 0,Y 342.725,Z 1007.845,A -85,B 0,C 180,E1 13245.371,E2 13245.371} C_VEL
LIN {X 0,Y 343.13,Z 1005.488,A -85,B 0,C 180,E1 13246.666,E2 13246.666} C_VEL
LIN {X 0,Y 342.385,Z 1002.939,A -85,B 0,C 180,E1 13248.059,E2 13248.059} C_VEL
LIN {X 0,Y 337.588,Z 995.225,A -85,B 0,C 180,E1 13251.856,E2 13251.856} C_VEL
LIN {X 0,Y 337.693,Z 994.409,A -85,B 0,C 180,E1 13252.203,E2 13252.203} C_VEL
LIN {X 0,Y 343.355,Z 974.853,A -85,B 0,C 180,E1 13259.017,E2 13259.017} C_VEL
LIN {X 0,Y 351.683,Z 950.148,A -85,B 0,C 180,E1 13265.267,E2 13265.267} C_VEL
LIN {X 0,Y 361.912,Z 921.264,A -85,B 0,C 180,E1 13270.646,E2 13270.646} C_VEL
LIN {X 0,Y 373.52,Z 887.017,A -85,B 0,C 180,E1 13275.314,E2 13275.314} C_VEL
LIN {X 0,Y 384.875,Z 849.388,A -85,B 0,C 180,E1 13278.993,E2 13278.993} C_VEL
LIN {X 0,Y 395.045,Z 808.309,A -85,B 0,C 180,E1 13281.773,E2 13281.773} C_VEL
LIN {X 0,Y 396.472,Z 799.191,A -85,B 0,C 180,E1 13282.336,E2 13282.336} C_VEL
LIN {X 0,Y 384.865,Z 771.06,A -85,B 0,C 180,E1 13286.954,E2 13286.954} C_VEL
LIN {X 0,Y 371.072,Z 745.448,A -85,B 0,C 180,E1 13292.261,E2 13292.261} C_VEL
LIN {X 0,Y 359.049,Z 727.133,A -85,B 0,C 180,E1 13297.366,E2 13297.366} C_VEL
LIN {X 0,Y 352.616,Z 718.752,A -85,B 0,C 180,E1 13300.559,E2 13300.559} C_VEL
LIN {X 0,Y 349.109,Z 713.481,A -85,B 0,C 180,E1 13302.586,E2 13302.586} C_VEL
LIN {X 0,Y 344.917,Z 707.725,A -85,B 0,C 180,E1 13305.376,E2 13305.376} C_VEL
LIN {X 0,Y 339.529,Z 701.266,A -85,B 0,C 180,E1 13310.044,E2 13310.044} C_VEL
LIN {X 0,Y 338.828,Z 699.137,A -85,B 0,C 180,E1 13310.997,E2 13310.997} C_VEL
LIN {X 0,Y 334.818,Z 696.115,A -85,B 0,C 180,E1 13320.872,E2 13320.872} C_VEL
LIN {X 0,Y 339.272,Z 699.921,A -85,B 0,C 180,E1 13330.032,E2 13330.032} C_VEL
LIN {X 0,Y 342.245,Z 705.333,A -85,B 0,C 180,E1 13333.096,E2 13333.096} C_VEL
LIN {X 0,Y 345.032,Z 707.744,A -85,B 0,C 180,E1 13335.18,E2 13335.18} C_VEL
LIN {X 0,Y 349.429,Z 713.676,A -85,B 0,C 180,E1 13338.117,E2 13338.117} C_VEL
LIN {X 0,Y 359.998,Z 729.034,A -85,B 0,C 180,E1 13343.787,E2 13343.787} C_VEL
LIN {X 0,Y 371.92,Z 748.746,A -85,B 0,C 180,E1 13349.149,E2 13349.149} C_VEL
LIN {X 0,Y 382.774,Z 770.882,A -85,B 0,C 180,E1 13353.832,E2 13353.832} C_VEL
LIN {X 0,Y 392.609,Z 797.782,A -85,B 0,C 180,E1 13358.515,E2 13358.515} C_VEL
LIN {X 0,Y 393.307,Z 802.629,A -85,B 0,C 180,E1 13359.154,E2 13359.154} C_VEL
LIN {X 0,Y 383.747,Z 839.055,A -85,B 0,C 180,E1 13361.955,E2 13361.955} C_VEL
LIN {X 0,Y 372.897,Z 873.556,A -85,B 0,C 180,E1 13365.64,E2 13365.64} C_VEL
LIN {X 0,Y 361.625,Z 905.442,A -85,B 0,C 180,E1 13370.319,E2 13370.319} C_VEL
LIN {X 0,Y 351.245,Z 933.313,A -85,B 0,C 180,E1 13375.917,E2 13375.917} C_VEL
LIN {X 0,Y 343.018,Z 956.274,A -85,B 0,C 180,E1 13382.266,E2 13382.266} C_VEL
LIN {X 0,Y 337.381,Z 974.676,A -85,B 0,C 180,E1 13389.474,E2 13389.474} C_VEL
LIN {X 0,Y 334.556,Z 987.191,A -85,B 0,C 180,E1 13396.921,E2 13396.921} C_VEL
LIN {X 0,Y 333.81,Z 992.559,A -85,B 0,C 180,E1 13402.179,E2 13402.179} C_VEL
LIN {X 0,Y 333.586,Z 995.192,A -85,B 0,C 180,E1 13407.398,E2 13407.398} C_VEL
LIN {X 0,Y 333.51,Z 994.975,A -85,B 0,C 180,E1 13413.121,E2 13413.121} C_VEL
LIN {X 0,Y 333.913,Z 991.319,A -85,B 0,C 180,E1 13419.131,E2 13419.131} C_VEL
LIN {X 0,Y 335.322,Z 983.272,A -85,B 0,C 180,E1 13425.718,E2 13425.718} C_VEL
LIN {X 0,Y 338.942,Z 968.904,A -85,B 0,C 180,E1 13433.008,E2 13433.008} C_VEL
LIN {X 0,Y 345.91,Z 947.833,A -85,B 0,C 180,E1 13440.222,E2 13440.222} C_VEL
LIN {X 0,Y 355.673,Z 921.474,A -85,B 0,C 180,E1 13446.581,E2 13446.581} C_VEL
LIN {X 0,Y 366.76,Z 891.214,A -85,B 0,C 180,E1 13451.863,E2 13451.863} C_VEL
LIN {X 0,Y 378.452,Z 856.611,A -85,B 0,C 180,E1 13456.224,E2 13456.224} C_VEL
LIN {X 0,Y 389.444,Z 818.162,A -85,B 0,C 180,E1 13459.683,E2 13459.683} C_VEL
LIN {X 0,Y 393.416,Z 800.703,A -85,B 0,C 180,E1 13460.922,E2 13460.922} C_VEL
LIN {X 0,Y 384.166,Z 774.232,A -85,B 0,C 180,E1 13465.434,E2 13465.434} C_VEL
LIN {X 0,Y 372.133,Z 749.317,A -85,B 0,C 180,E1 13470.622,E2 13470.622} C_VEL
LIN {X 0,Y 361.182,Z 731.252,A -85,B 0,C 180,E1 13475.474,E2 13475.474} C_VEL
LIN {X 0,Y 353.398,Z 719.815,A -85,B 0,C 180,E1 13479.392,E2 13479.392} C_VEL
LIN {X 0,Y 348.903,Z 713.36,A -85,B 0,C 180,E1 13481.998,E2 13481.998} C_VEL
LIN {X 0,Y 344.813,Z 706.952,A -85,B 0,C 180,E1 13484.814,E2 13484.814} C_VEL
LIN {X 0,Y 339.671,Z 701.445,A -85,B 0,C 180,E1 13489.133,E2 13489.133} C_VEL
LIN {X 0,Y 338.691,Z 699.09,A -85,B 0,C 180,E1 13490.357,E2 13490.357} C_VEL
LIN {X 0,Y 334.645,Z 695.735,A -85,B 0,C 180,E1 13500.679,E2 13500.679} C_VEL
LIN {X 0,Y 339.245,Z 699.913,A -85,B 0,C 180,E1 13509.721,E2 13509.721} C_VEL
LIN {X 0,Y 342.114,Z 705.254,A -85,B 0,C 180,E1 13512.652,E2 13512.652} C_VEL
LIN {X 0,Y 345.082,Z 707.983,A -85,B 0,C 180,E1 13514.861,E2 13514.861} C_VEL
LIN {X 0,Y 349.674,Z 713.814,A -85,B 0,C 180,E1 13517.81,E2 13517.81} C_VEL
LIN {X 0,Y 360.97,Z 730.087,A -85,B 0,C 180,E1 13523.568,E2 13523.568} C_VEL
LIN {X 0,Y 372.72,Z 748.458,A -85,B 0,C 180,E1 13528.43,E2 13528.43} C_VEL
LIN {X 0,Y 386.167,Z 773.842,A -85,B 0,C 180,E1 13533.57,E2 13533.57} C_VEL
LIN {X 0,Y 396.412,Z 799.224,A -85,B 0,C 180,E1 13537.671,E2 13537.671} C_VEL
LIN {X 0,Y 387.368,Z 840.14,A -85,B 0,C 180,E1 13540.29,E2 13540.29} C_VEL
LIN {X 0,Y 376.577,Z 877.525,A -85,B 0,C 180,E1 13543.638,E2 13543.638} C_VEL
LIN {X 0,Y 364.994,Z 912.547,A -85,B 0,C 180,E1 13548.018,E2 13548.018} C_VEL
LIN {X 0,Y 353.834,Z 944.232,A -85,B 0,C 180,E1 13553.484,E2 13553.484} C_VEL
LIN {X 0,Y 344.387,Z 971.516,A -85,B 0,C 180,E1 13559.994,E2 13559.994} C_VEL
LIN {X 0,Y 338.207,Z 992.375,A -85,B 0,C 180,E1 13566.939,E2 13566.939} C_VEL
LIN {X 0,Y 334.926,Z 1007.541,A -85,B 0,C 180,E1 13574.262,E2 13574.262} C_VEL
LIN {X 0,Y 333.8,Z 1016.081,A -85,B 0,C 180,E1 13580.866,E2 13580.866} C_VEL
LIN {X 0,Y 333.607,Z 1020.175,A -85,B 0,C 180,E1 13587.399,E2 13587.399} C_VEL
LIN {X 0,Y 333.508,Z 1020.07,A -85,B 0,C 180,E1 13592.872,E2 13592.872} C_VEL
LIN {X 0,Y 333.812,Z 1016.082,A -85,B 0,C 180,E1 13599.135,E2 13599.135} C_VEL
LIN {X 0,Y 334.93,Z 1007.542,A -85,B 0,C 180,E1 13605.738,E2 13605.738} C_VEL
LIN {X 0,Y 337.693,Z 994.409,A -85,B 0,C 180,E1 13612.203,E2 13612.203} C_VEL
LIN {X 0,Y 335.649,Z 987.978,A -85,B 0,C 180,E1 13614.958,E2 13614.958} C_VEL
LIN {X 0,Y 334.1,Z 980.872,A -85,B 0,C 180,E1 13617.696,E2 13617.696} C_VEL
LIN {X 0,Y 342.206,Z 957.314,A -85,B 0,C 180,E1 13624.342,E2 13624.342} C_VEL
LIN {X 0,Y 352.65,Z 929.303,A -85,B 0,C 180,E1 13630.093,E2 13630.093} C_VEL
LIN {X 0,Y 364.271,Z 897.008,A -85,B 0,C 180,E1 13634.96,E2 13634.96} C_VEL
LIN {X 0,Y 376.08,Z 861.113,A -85,B 0,C 180,E1 13638.863,E2 13638.863} C_VEL
LIN {X 0,Y 386.554,Z 823.634,A -85,B 0,C 180,E1 13641.757,E2 13641.757} C_VEL
LIN {X 0,Y 391.061,Z 803.356,A -85,B 0,C 180,E1 13642.956,E2 13642.956} C_VEL
LIN {X 0,Y 380.143,Z 775.698,A -85,B 0,C 180,E1 13647.666,E2 13647.666} C_VEL
LIN {X 0,Y 367.713,Z 751.751,A -85,B 0,C 180,E1 13652.817,E2 13652.817} C_VEL
LIN {X 0,Y 356.485,Z 733.921,A -85,B 0,C 180,E1 13657.934,E2 13657.934} C_VEL
LIN {X 0,Y 347.355,Z 720.914,A -85,B 0,C 180,E1 13662.966,E2 13662.966} C_VEL
LIN {X 0,Y 343.146,Z 714.61,A -85,B 0,C 180,E1 13665.951,E2 13665.951} C_VEL
LIN {X 0,Y 338.326,Z 709.154,A -85,B 0,C 180,E1 13670.253,E2 13670.253} C_VEL
LIN {X 0,Y 337.308,Z 706.814,A -85,B 0,C 180,E1 13671.606,E2 13671.606} C_VEL
LIN {X 0,Y 333.855,Z 703.959,A -85,B 0,C 180,E1 13680.875,E2 13680.875} C_VEL
LIN {X 0,Y 337.992,Z 707.759,A -85,B 0,C 180,E1 13689.729,E2 13689.729} C_VEL
LIN {X 0,Y 341.636,Z 713.552,A -85,B 0,C 180,E1 13693.446,E2 13693.446} C_VEL
LIN {X 0,Y 343.613,Z 715.867,A -85,B 0,C 180,E1 13695.013,E2 13695.013} C_VEL
LIN {X 0,Y 349.089,Z 723.832,A -85,B 0,C 180,E1 13698.728,E2 13698.728} C_VEL
LIN {X 0,Y 357.3,Z 735.886,A -85,B 0,C 180,E1 13703.315,E2 13703.315} C_VEL
LIN {X 0,Y 368.843,Z 756.082,A -85,B 0,C 180,E1 13708.911,E2 13708.911} C_VEL
LIN {X 0,Y 380.009,Z 780.574,A -85,B 0,C 180,E1 13714.112,E2 13714.112} C_VEL
LIN {X 0,Y 387.755,Z 804.009,A -85,B 0,C 180,E1 13718.249,E2 13718.249} C_VEL
LIN {X 0,Y 377.063,Z 843.928,A -85,B 0,C 180,E1 13721.47,E2 13721.47} C_VEL
LIN {X 0,Y 365.344,Z 878.98,A -85,B 0,C 180,E1 13725.417,E2 13725.417} C_VEL
LIN {X 0,Y 353.649,Z 910.208,A -85,B 0,C 180,E1 13730.278,E2 13730.278} C_VEL
LIN {X 0,Y 343.378,Z 936.478,A -85,B 0,C 180,E1 13735.868,E2 13735.868} C_VEL
LIN {X 0,Y 335.159,Z 958.282,A -85,B 0,C 180,E1 13742.214,E2 13742.214} C_VEL
LIN {X 0,Y 329.56,Z 975.732,A -85,B 0,C 180,E1 13749.372,E2 13749.372} C_VEL
LIN {X 0,Y 326.768,Z 987.49,A -85,B 0,C 180,E1 13756.604,E2 13756.604} C_VEL
LIN {X 0,Y 325.93,Z 992.857,A -85,B 0,C 180,E1 13761.989,E2 13761.989} C_VEL
LIN {X 0,Y 325.7,Z 995.488,A -85,B 0,C 180,E1 13767.335,E2 13767.335} C_VEL
LIN {X 0,Y 325.672,Z 995.466,A -85,B 0,C 180,E1 13772.664,E2 13772.664} C_VEL
LIN {X 0,Y 326.065,Z 991.618,A -85,B 0,C 180,E1 13779.353,E2 13779.353} C_VEL
LIN {X 0,Y 327.59,Z 983.575,A -85,B 0,C 180,E1 13786.099,E2 13786.099} C_VEL
LIN {X 0,Y 331.486,Z 969.21,A -85,B 0,C 180,E1 13793.557,E2 13793.557} C_VEL
LIN {X 0,Y 338.908,Z 948.14,A -85,B 0,C 180,E1 13800.914,E2 13800.914} C_VEL
LIN {X 0,Y 349.165,Z 921.782,A -85,B 0,C 180,E1 13807.378,E2 13807.378} C_VEL
LIN {X 0,Y 360.992,Z 890.848,A -85,B 0,C 180,E1 13812.822,E2 13812.822} C_VEL
LIN {X 0,Y 373.147,Z 856.22,A -85,B 0,C 180,E1 13817.189,E2 13817.189} C_VEL
LIN {X 0,Y 384.27,Z 818.714,A -85,B 0,C 180,E1 13820.572,E2 13820.572} C_VEL
LIN {X 0,Y 387.834,Z 804.536,A -85,B 0,C 180,E1 13821.573,E2 13821.573} C_VEL
LIN {X 0,Y 378.823,Z 777.7,A -85,B 0,C 180,E1 13826.332,E2 13826.332} C_VEL
LIN {X 0,Y 366.79,Z 752.034,A -85,B 0,C 180,E1 13831.953,E2 13831.953} C_VEL
LIN {X 0,Y 355.723,Z 733.71,A -85,B 0,C 180,E1 13837.321,E2 13837.321} C_VEL
LIN {X 0,Y 347.279,Z 720.952,A -85,B 0,C 180,E1 13842.239,E2 13842.239} C_VEL
LIN {X 0,Y 342.375,Z 714.013,A -85,B 0,C 180,E1 13845.768,E2 13845.768} C_VEL
LIN {X 0,Y 338.074,Z 708.108,A -85,B 0,C 180,E1 13849.851,E2 13849.851} C_VEL
LIN {X 0,Y 336.639,Z 706.535,A -85,B 0,C 180,E1 13851.602,E2 13851.602} C_VEL
LIN {X 0,Y 333.685,Z 703.551,A -85,B 0,C 180,E1 13860.681,E2 13860.681} C_VEL
LIN {X 0,Y 337.97,Z 707.765,A -85,B 0,C 180,E1 13869.432,E2 13869.432} C_VEL
LIN {X 0,Y 341.325,Z 713.339,A -85,B 0,C 180,E1 13872.819,E2 13872.819} C_VEL
LIN {X 0,Y 343.563,Z 715.623,A -85,B 0,C 180,E1 13874.52,E2 13874.52} C_VEL
LIN {X 0,Y 349.27,Z 723.879,A -85,B 0,C 180,E1 13878.321,E2 13878.321} C_VEL
LIN {X 0,Y 358.131,Z 736.405,A -85,B 0,C 180,E1 13882.942,E2 13882.942} C_VEL
LIN {X 0,Y 369.883,Z 755.79,A -85,B 0,C 180,E1 13888.168,E2 13888.168} C_VEL
LIN {X 0,Y 382.622,Z 781.091,A -85,B 0,C 180,E1 13893.348,E2 13893.348} C_VEL
LIN {X 0,Y 390.93,Z 803.06,A -85,B 0,C 180,E1 13897.008,E2 13897.008} C_VEL
LIN {X 0,Y 381.205,Z 843.256,A -85,B 0,C 180,E1 13899.632,E2 13899.632} C_VEL
LIN {X 0,Y 370.133,Z 879.784,A -85,B 0,C 180,E1 13903.014,E2 13903.014} C_VEL
LIN {X 0,Y 358.187,Z 914.222,A -85,B 0,C 180,E1 13907.443,E2 13907.443} C_VEL
LIN {X 0,Y 346.49,Z 945.823,A -85,B 0,C 180,E1 13913.079,E2 13913.079} C_VEL
LIN {X 0,Y 337.44,Z 970.839,A -85,B 0,C 180,E1 13919.187,E2 13919.187} C_VEL
LIN {X 0,Y 330.785,Z 991.776,A -85,B 0,C 180,E1 13926.267,E2 13926.267} C_VEL
LIN {X 0,Y 327.139,Z 1007.236,A -85,B 0,C 180,E1 13933.878,E2 13933.878} C_VEL
LIN {X 0,Y 325.907,Z 1015.781,A -85,B 0,C 180,E1 13940.643,E2 13940.643} C_VEL
LIN {X 0,Y 325.72,Z 1019.879,A -85,B 0,C 180,E1 13947.336,E2 13947.336} C_VEL
LIN {X 0,Y 325.653,Z 1019.877,A -85,B 0,C 180,E1 13952.665,E2 13952.665} C_VEL
LIN {X 0,Y 325.919,Z 1015.783,A -85,B 0,C 180,E1 13959.358,E2 13959.358} C_VEL
LIN {X 0,Y 327.144,Z 1007.239,A -85,B 0,C 180,E1 13966.123,E2 13966.123} C_VEL
LIN {X 0,Y 330.804,Z 991.763,A -85,B 0,C 180,E1 13973.74,E2 13973.74} C_VEL
LIN {X 0,Y 334.1,Z 980.872,A -85,B 0,C 180,E1 13977.696,E2 13977.696} C_VEL
LIN {X 0,Y 332.963,Z 973.281,A -85,B 0,C 180,E1 13980.406,E2 13980.406} C_VEL
LIN {X 0,Y 332.366,Z 965.038,A -85,B 0,C 180,E1 13983.073,E2 13983.073} C_VEL
LIN {X 0,Y 342.77,Z 938.107,A -85,B 0,C 180,E1 13989.276,E2 13989.276} C_VEL
LIN {X 0,Y 354.85,Z 906.952,A -85,B 0,C 180,E1 13994.478,E2 13994.478} C_VEL
LIN {X 0,Y 366.44,Z 874.258,A -85,B 0,C 180,E1 13998.488,E2 13998.488} C_VEL
LIN {X 0,Y 377.853,Z 837.209,A -85,B 0,C 180,E1 14001.763,E2 14001.763} C_VEL
LIN {X 0,Y 385.465,Z 806.614,A -85,B 0,C 180,E1 14003.726,E2 14003.726} C_VEL
LIN {X 0,Y 375.022,Z 779.423,A -85,B 0,C 180,E1 14008.584,E2 14008.584} C_VEL
LIN {X 0,Y 363.419,Z 756.643,A -85,B 0,C 180,E1 14013.724,E2 14013.724} C_VEL
LIN {X 0,Y 353.687,Z 740.619,A -85,B 0,C 180,E1 14018.494,E2 14018.494} C_VEL
LIN {X 0,Y 345.125,Z 727.956,A -85,B 0,C 180,E1 14023.591,E2 14023.591} C_VEL
LIN {X 0,Y 340.635,Z 721.582,A -85,B 0,C 180,E1 14026.991,E2 14026.991} C_VEL
LIN {X 0,Y 336.798,Z 715.877,A -85,B 0,C 180,E1 14030.942,E2 14030.942} C_VEL
LIN {X 0,Y 335.131,Z 714.088,A -85,B 0,C 180,E1 14033.184,E2 14033.184} C_VEL
LIN {X 0,Y 332.94,Z 711.854,A -85,B 0,C 180,E1 14041.451,E2 14041.451} C_VEL
LIN {X 0,Y 336.665,Z 715.489,A -85,B 0,C 180,E1 14049.434,E2 14049.434} C_VEL
LIN {X 0,Y 340.709,Z 721.62,A -85,B 0,C 180,E1 14053.647,E2 14053.647} C_VEL
LIN {X 0,Y 346.908,Z 731.132,A -85,B 0,C 180,E1 14058.356,E2 14058.356} C_VEL
LIN {X 0,Y 354.836,Z 743.426,A -85,B 0,C 180,E1 14063.071,E2 14063.071} C_VEL
LIN {X 0,Y 365.233,Z 762.512,A -85,B 0,C 180,E1 14068.469,E2 14068.469} C_VEL
LIN {X 0,Y 375.342,Z 786.053,A -85,B 0,C 180,E1 14073.617,E2 14073.617} C_VEL
LIN {X 0,Y 382.207,Z 807.932,A -85,B 0,C 180,E1 14077.6,E2 14077.6} C_VEL
LIN {X 0,Y 371.229,Z 846.11,A -85,B 0,C 180,E1 14080.721,E2 14080.721} C_VEL
LIN {X 0,Y 358.708,Z 881.888,A -85,B 0,C 180,E1 14084.858,E2 14084.858} C_VEL
LIN {X 0,Y 345.975,Z 914.213,A -85,B 0,C 180,E1 14090.102,E2 14090.102} C_VEL
LIN {X 0,Y 334.716,Z 941.677,A -85,B 0,C 180,E1 14096.349,E2 14096.349} C_VEL
LIN {X 0,Y 326.382,Z 962.919,A -85,B 0,C 180,E1 14103.108,E2 14103.108} C_VEL
LIN {X 0,Y 321.027,Z 979.506,A -85,B 0,C 180,E1 14110.722,E2 14110.722} C_VEL
LIN {X 0,Y 318.604,Z 989.472,A -85,B 0,C 180,E1 14117.794,E2 14117.794} C_VEL
LIN {X 0,Y 317.86,Z 994.804,A -85,B 0,C 180,E1 14124.533,E2 14124.533} C_VEL
LIN {X 0,Y 317.839,Z 996.101,A -85,B 0,C 180,E1 14129.999,E2 14129.999} C_VEL
LIN {X 0,Y 317.791,Z 994.761,A -85,B 0,C 180,E1 14135.467,E2 14135.467} C_VEL
LIN {X 0,Y 318.621,Z 989.355,A -85,B 0,C 180,E1 14142.219,E2 14142.219} C_VEL
LIN {X 0,Y 321.194,Z 978.876,A -85,B 0,C 180,E1 14149.518,E2 14149.518} C_VEL
LIN {X 0,Y 326.501,Z 962.677,A -85,B 0,C 180,E1 14156.88,E2 14156.88} C_VEL
LIN {X 0,Y 335.172,Z 940.734,A -85,B 0,C 180,E1 14163.795,E2 14163.795} C_VEL
LIN {X 0,Y 346.244,Z 913.477,A -85,B 0,C 180,E1 14169.94,E2 14169.94} C_VEL
LIN {X 0,Y 358.927,Z 881.013,A -85,B 0,C 180,E1 14175.17,E2 14175.17} C_VEL
LIN {X 0,Y 371.77,Z 844.25,A -85,B 0,C 180,E1 14179.35,E2 14179.35} C_VEL
LIN {X 0,Y 382.023,Z 807.089,A -85,B 0,C 180,E1 14182.435,E2 14182.435} C_VEL
LIN {X 0,Y 373.5,Z 781.258,A -85,B 0,C 180,E1 14187.245,E2 14187.245} C_VEL
LIN {X 0,Y 362.788,Z 757.845,A -85,B 0,C 180,E1 14192.607,E2 14192.607} C_VEL
LIN {X 0,Y 353.011,Z 740.539,A -85,B 0,C 180,E1 14197.802,E2 14197.802} C_VEL
LIN {X 0,Y 344.799,Z 727.883,A -85,B 0,C 180,E1 14202.932,E2 14202.932} C_VEL
LIN {X 0,Y 340.642,Z 721.514,A -85,B 0,C 180,E1 14206.186,E2 14206.186} C_VEL
LIN {X 0,Y 336.636,Z 715.433,A -85,B 0,C 180,E1 14210.298,E2 14210.298} C_VEL
LIN {X 0,Y 332.703,Z 711.2,A -85,B 0,C 180,E1 14220.006,E2 14220.006} C_VEL
LIN {X 0,Y 336.738,Z 715.661,A -85,B 0,C 180,E1 14229.182,E2 14229.182} C_VEL
LIN {X 0,Y 340.68,Z 721.527,A -85,B 0,C 180,E1 14233.17,E2 14233.17} C_VEL
LIN {X 0,Y 347.354,Z 731.214,A -85,B 0,C 180,E1 14237.933,E2 14237.933} C_VEL
LIN {X 0,Y 356.14,Z 744.466,A -85,B 0,C 180,E1 14242.829,E2 14242.829} C_VEL
LIN {X 0,Y 367.881,Z 764.625,A -85,B 0,C 180,E1 14248.285,E2 14248.285} C_VEL
LIN {X 0,Y 379.753,Z 790.541,A -85,B 0,C 180,E1 14253.566,E2 14253.566} C_VEL
LIN {X 0,Y 385.419,Z 806.572,A -85,B 0,C 180,E1 14256.279,E2 14256.279} C_VEL
LIN {X 0,Y 375.123,Z 846.305,A -85,B 0,C 180,E1 14258.948,E2 14258.948} C_VEL
LIN {X 0,Y 363.724,Z 882.029,A -85,B 0,C 180,E1 14262.364,E2 14262.364} C_VEL
LIN {X 0,Y 351.558,Z 915.446,A -85,B 0,C 180,E1 14266.778,E2 14266.778} C_VEL
LIN {X 0,Y 339.893,Z 945.477,A -85,B 0,C 180,E1 14272.23,E2 14272.23} C_VEL
LIN {X 0,Y 330.289,Z 970.86,A -85,B 0,C 180,E1 14278.558,E2 14278.558} C_VEL
LIN {X 0,Y 323.152,Z 991.923,A -85,B 0,C 180,E1 14285.873,E2 14285.873} C_VEL
LIN {X 0,Y 319.353,Z 1006.931,A -85,B 0,C 180,E1 14293.474,E2 14293.474} C_VEL
LIN {X 0,Y 318.016,Z 1015.481,A -85,B 0,C 180,E1 14300.408,E2 14300.408} C_VEL
LIN {X 0,Y 317.839,Z 1019.583,A -85,B 0,C 180,E1 14307.27,E2 14307.27} C_VEL
LIN {X 0,Y 317.748,Z 1019.58,A -85,B 0,C 180,E1 14312.732,E2 14312.732} C_VEL
LIN {X 0,Y 318.028,Z 1015.483,A -85,B 0,C 180,E1 14319.592,E2 14319.592} C_VEL
LIN {X 0,Y 319.355,Z 1006.935,A -85,B 0,C 180,E1 14326.527,E2 14326.527} C_VEL
LIN {X 0,Y 323.162,Z 991.922,A -85,B 0,C 180,E1 14334.131,E2 14334.131} C_VEL
LIN {X 0,Y 330.214,Z 970.935,A -85,B 0,C 180,E1 14341.428,E2 14341.428} C_VEL
LIN {X 0,Y 332.366,Z 965.038,A -85,B 0,C 180,E1 14343.073,E2 14343.073} C_VEL
LIN {X 0,Y 332.338,Z 956.293,A -85,B 0,C 180,E1 14345.693,E2 14345.693} C_VEL
LIN {X 0,Y 332.734,Z 946.93,A -85,B 0,C 180,E1 14348.248,E2 14348.248} C_VEL
LIN {X 0,Y 344.29,Z 918.429,A -85,B 0,C 180,E1 14353.641,E2 14353.641} C_VEL
LIN {X 0,Y 356.875,Z 885.636,A -85,B 0,C 180,E1 14358.169,E2 14358.169} C_VEL
LIN {X 0,Y 369.481,Z 848.236,A -85,B 0,C 180,E1 14361.855,E2 14361.855} C_VEL
LIN {X 0,Y 379.772,Z 809.558,A -85,B 0,C 180,E1 14364.583,E2 14364.583} C_VEL
LIN {X 0,Y 370.384,Z 784.3,A -85,B 0,C 180,E1 14369.267,E2 14369.267} C_VEL
LIN {X 0,Y 359.465,Z 761.859,A -85,B 0,C 180,E1 14374.542,E2 14374.542} C_VEL
LIN {X 0,Y 349.593,Z 745.274,A -85,B 0,C 180,E1 14379.807,E2 14379.807} C_VEL
LIN {X 0,Y 343.042,Z 735.213,A -85,B 0,C 180,E1 14384.065,E2 14384.065} C_VEL
LIN {X 0,Y 338.928,Z 729.061,A -85,B 0,C 180,E1 14387.417,E2 14387.417} C_VEL
LIN {X 0,Y 335.261,Z 722.954,A -85,B 0,C 180,E1 14391.473,E2 14391.473} C_VEL
LIN {X 0,Y 331.799,Z 719.567,A -85,B 0,C 180,E1 14400.647,E2 14400.647} C_VEL
LIN {X 0,Y 335.272,Z 723.25,A -85,B 0,C 180,E1 14409.169,E2 14409.169} C_VEL
LIN {X 0,Y 339.235,Z 729.355,A -85,B 0,C 180,E1 14413.543,E2 14413.543} C_VEL
LIN {X 0,Y 345.037,Z 738.985,A -85,B 0,C 180,E1 14418.21,E2 14418.21} C_VEL
LIN {X 0,Y 352.309,Z 751.004,A -85,B 0,C 180,E1 14422.852,E2 14422.852} C_VEL
LIN {X 0,Y 362.327,Z 770.343,A -85,B 0,C 180,E1 14428.427,E2 14428.427} C_VEL
LIN {X 0,Y 371.71,Z 794.53,A -85,B 0,C 180,E1 14433.698,E2 14433.698} C_VEL
LIN {X 0,Y 376.387,Z 812.11,A -85,B 0,C 180,E1 14436.931,E2 14436.931} C_VEL
LIN {X 0,Y 365.534,Z 847.847,A -85,B 0,C 180,E1 14439.914,E2 14439.914} C_VEL
LIN {X 0,Y 352.753,Z 882.934,A -85,B 0,C 180,E1 14444.032,E2 14444.032} C_VEL
LIN {X 0,Y 339.794,Z 914.516,A -85,B 0,C 180,E1 14449.226,E2 14449.226} C_VEL
LIN {X 0,Y 327.948,Z 941.981,A -85,B 0,C 180,E1 14455.558,E2 14455.558} C_VEL
LIN {X 0,Y 319.127,Z 963.223,A -85,B 0,C 180,E1 14462.445,E2 14462.445} C_VEL
LIN {X 0,Y 313.399,Z 979.808,A -85,B 0,C 180,E1 14470.233,E2 14470.233} C_VEL
LIN {X 0,Y 310.74,Z 990.093,A -85,B 0,C 180,E1 14477.784,E2 14477.784} C_VEL
LIN {X 0,Y 309.962,Z 995.102,A -85,B 0,C 180,E1 14484.393,E2 14484.393} C_VEL
LIN {X 0,Y 309.943,Z 996.397,A -85,B 0,C 180,E1 14489.999,E2 14489.999} C_VEL
LIN {X 0,Y 309.897,Z 995.059,A -85,B 0,C 180,E1 14495.607,E2 14495.607} C_VEL
LIN {X 0,Y 310.954,Z 988.942,A -85,B 0,C 180,E1 14503.201,E2 14503.201} C_VEL
LIN {X 0,Y 313.84,Z 978.336,A -85,B 0,C 180,E1 14510.473,E2 14510.473} C_VEL
LIN {X 0,Y 319.23,Z 962.985,A -85,B 0,C 180,E1 14517.544,E2 14517.544} C_VEL
LIN {X 0,Y 328.673,Z 940.402,A -85,B 0,C 180,E1 14524.755,E2 14524.755} C_VEL
LIN {X 0,Y 340.114,Z 913.673,A -85,B 0,C 180,E1 14530.837,E2 14530.837} C_VEL
LIN {X 0,Y 353.275,Z 881.317,A -85,B 0,C 180,E1 14536.1,E2 14536.1} C_VEL
LIN {X 0,Y 366.575,Z 844.558,A -85,B 0,C 180,E1 14540.305,E2 14540.305} C_VEL
LIN {X 0,Y 376.413,Z 810.732,A -85,B 0,C 180,E1 14543.132,E2 14543.132} C_VEL
LIN {X 0,Y 368.253,Z 784.962,A -85,B 0,C 180,E1 14548.144,E2 14548.144} C_VEL
LIN {X 0,Y 358.299,Z 762.503,A -85,B 0,C 180,E1 14553.571,E2 14553.571} C_VEL
LIN {X 0,Y 349.852,Z 746.997,A -85,B 0,C 180,E1 14558.426,E2 14558.426} C_VEL
LIN {X 0,Y 342.547,Z 735.033,A -85,B 0,C 180,E1 14563.395,E2 14563.395} C_VEL
LIN {X 0,Y 338.787,Z 729.013,A -85,B 0,C 180,E1 14566.603,E2 14566.603} C_VEL
LIN {X 0,Y 334.509,Z 722.214,A -85,B 0,C 180,E1 14571.548,E2 14571.548} C_VEL
LIN {X 0,Y 331.645,Z 719.226,A -85,B 0,C 180,E1 14580.66,E2 14580.66} C_VEL
LIN {X 0,Y 335.363,Z 723.413,A -85,B 0,C 180,E1 14588.933,E2 14588.933} C_VEL
LIN {X 0,Y 339.561,Z 729.412,A -85,B 0,C 180,E1 14593.214,E2 14593.214} C_VEL
LIN {X 0,Y 345.647,Z 739.31,A -85,B 0,C 180,E1 14597.86,E2 14597.86} C_VEL
LIN {X 0,Y 354.298,Z 752.828,A -85,B 0,C 180,E1 14602.872,E2 14602.872} C_VEL
LIN {X 0,Y 364.821,Z 772.418,A -85,B 0,C 180,E1 14608.138,E2 14608.138} C_VEL
LIN {X 0,Y 375.55,Z 797.132,A -85,B 0,C 180,E1 14613.256,E2 14613.256} C_VEL
LIN {X 0,Y 379.596,Z 811.328,A -85,B 0,C 180,E1 14615.596,E2 14615.596} C_VEL
LIN {X 0,Y 368.434,Z 851.521,A -85,B 0,C 180,E1 14618.421,E2 14618.421} C_VEL
LIN {X 0,Y 355.551,Z 889.337,A -85,B 0,C 180,E1 14622.278,E2 14622.278} C_VEL
LIN {X 0,Y 342.408,Z 923.251,A -85,B 0,C 180,E1 14627.155,E2 14627.155} C_VEL
LIN {X 0,Y 330.202,Z 953.15,A -85,B 0,C 180,E1 14633.162,E2 14633.162} C_VEL
LIN {X 0,Y 320.246,Z 978.291,A -85,B 0,C 180,E1 14640.237,E2 14640.237} C_VEL
LIN {X 0,Y 313.805,Z 997.682,A -85,B 0,C 180,E1 14648.042,E2 14648.042} C_VEL
LIN {X 0,Y 310.818,Z 1010.653,A -85,B 0,C 180,E1 14655.904,E2 14655.904} C_VEL
LIN {X 0,Y 310.033,Z 1016.425,A -85,B 0,C 180,E1 14661.576,E2 14661.576} C_VEL
LIN {X 0,Y 309.93,Z 1019.286,A -85,B 0,C 180,E1 14667.2,E2 14667.2} C_VEL
LIN {X 0,Y 309.842,Z 1019.284,A -85,B 0,C 180,E1 14672.801,E2 14672.801} C_VEL
LIN {X 0,Y 310.142,Z 1015.184,A -85,B 0,C 180,E1 14679.839,E2 14679.839} C_VEL
LIN {X 0,Y 311.597,Z 1006.632,A -85,B 0,C 180,E1 14686.951,E2 14686.951} C_VEL
LIN {X 0,Y 315.674,Z 991.639,A -85,B 0,C 180,E1 14694.73,E2 14694.73} C_VEL
LIN {X 0,Y 323.573,Z 969.616,A -85,B 0,C 180,E1 14702.496,E2 14702.496} C_VEL
LIN {X 0,Y 332.734,Z 946.93,A -85,B 0,C 180,E1 14708.248,E2 14708.248} C_VEL
LIN {X 0,Y 333.578,Z 937.078,A -85,B 0,C 180,E1 14710.743,E2 14710.743} C_VEL
LIN {X 0,Y 334.822,Z 926.631,A -85,B 0,C 180,E1 14713.147,E2 14713.147} C_VEL
LIN {X 0,Y 347.775,Z 894.932,A -85,B 0,C 180,E1 14717.974,E2 14717.974} C_VEL
LIN {X 0,Y 360.665,Z 859.762,A -85,B 0,C 180,E1 14721.822,E2 14721.822} C_VEL
LIN {X 0,Y 372.4,Z 821.58,A -85,B 0,C 180,E1 14724.748,E2 14724.748} C_VEL
LIN {X 0,Y 374.309,Z 813.964,A -85,B 0,C 180,E1 14725.225,E2 14725.225} C_VEL
LIN {X 0,Y 366.731,Z 791.609,A -85,B 0,C 180,E1 14729.462,E2 14729.462} C_VEL
LIN {X 0,Y 356.377,Z 768.933,A -85,B 0,C 180,E1 14734.856,E2 14734.856} C_VEL
LIN {X 0,Y 347.576,Z 753.338,A -85,B 0,C 180,E1 14739.851,E2 14739.851} C_VEL
LIN {X 0,Y 340.904,Z 742.5,A -85,B 0,C 180,E1 14744.458,E2 14744.458} C_VEL
LIN {X 0,Y 337.023,Z 736.472,A -85,B 0,C 180,E1 14747.839,E2 14747.839} C_VEL
LIN {X 0,Y 333.129,Z 729.817,A -85,B 0,C 180,E1 14752.815,E2 14752.815} C_VEL
LIN {X 0,Y 330.693,Z 727.458,A -85,B 0,C 180,E1 14761.305,E2 14761.305} C_VEL
LIN {X 0,Y 333.744,Z 731.026,A -85,B 0,C 180,E1 14768.964,E2 14768.964} C_VEL
LIN {X 0,Y 338.509,Z 739.193,A -85,B 0,C 180,E1 14774.398,E2 14774.398} C_VEL
LIN {X 0,Y 343.074,Z 747.107,A -85,B 0,C 180,E1 14778.235,E2 14778.235} C_VEL
LIN {X 0,Y 351.299,Z 761.38,A -85,B 0,C 180,E1 14783.673,E2 14783.673} C_VEL
LIN {X 0,Y 361.17,Z 783.451,A -85,B 0,C 180,E1 14789.612,E2 14789.612} C_VEL
LIN {X 0,Y 369.19,Z 807.855,A -85,B 0,C 180,E1 14794.77,E2 14794.77} C_VEL
LIN {X 0,Y 370.762,Z 815.495,A -85,B 0,C 180,E1 14796.166,E2 14796.166} C_VEL
LIN {X 0,Y 359.26,Z 851.422,A -85,B 0,C 180,E1 14799.274,E2 14799.274} C_VEL
LIN {X 0,Y 346.301,Z 885.307,A -85,B 0,C 180,E1 14803.374,E2 14803.374} C_VEL
LIN {X 0,Y 333.08,Z 916.075,A -85,B 0,C 180,E1 14808.569,E2 14808.569} C_VEL
LIN {X 0,Y 321.237,Z 942.285,A -85,B 0,C 180,E1 14814.733,E2 14814.733} C_VEL
LIN {X 0,Y 311.913,Z 963.528,A -85,B 0,C 180,E1 14821.752,E2 14821.752} C_VEL
LIN {X 0,Y 305.797,Z 980.11,A -85,B 0,C 180,E1 14829.721,E2 14829.721} C_VEL
LIN {X 0,Y 303.083,Z 989.671,A -85,B 0,C 180,E1 14836.771,E2 14836.771} C_VEL
LIN {X 0,Y 302.072,Z 995.399,A -85,B 0,C 180,E1 14844.246,E2 14844.246} C_VEL
LIN {X 0,Y 302.053,Z 996.693,A -85,B 0,C 180,E1 14849.999,E2 14849.999} C_VEL
LIN {X 0,Y 302.016,Z 995.357,A -85,B 0,C 180,E1 14855.754,E2 14855.754} C_VEL
LIN {X 0,Y 303.104,Z 989.544,A -85,B 0,C 180,E1 14863.255,E2 14863.255} C_VEL
LIN {X 0,Y 306.229,Z 978.643,A -85,B 0,C 180,E1 14871.005,E2 14871.005} C_VEL
LIN {X 0,Y 311.993,Z 963.294,A -85,B 0,C 180,E1 14878.239,E2 14878.239} C_VEL
LIN {X 0,Y 321.996,Z 940.711,A -85,B 0,C 180,E1 14885.583,E2 14885.583} C_VEL
LIN {X 0,Y 334.015,Z 913.981,A -85,B 0,C 180,E1 14891.747,E2 14891.747} C_VEL
LIN {X 0,Y 347.727,Z 881.623,A -85,B 0,C 180,E1 14897.058,E2 14897.058} C_VEL
LIN {X 0,Y 361.514,Z 844.852,A -85,B 0,C 180,E1 14901.283,E2 14901.283} C_VEL
LIN {X 0,Y 370.729,Z 813.965,A -85,B 0,C 180,E1 14903.934,E2 14903.934} C_VEL
LIN {X 0,Y 363.252,Z 789.207,A -85,B 0,C 180,E1 14908.96,E2 14908.96} C_VEL
LIN {X 0,Y 353.541,Z 766.098,A -85,B 0,C 180,E1 14914.808,E2 14914.808} C_VEL
LIN {X 0,Y 344.628,Z 749.373,A -85,B 0,C 180,E1 14920.52,E2 14920.52} C_VEL
LIN {X 0,Y 337.319,Z 736.852,A -85,B 0,C 180,E1 14926.544,E2 14926.544} C_VEL
LIN {X 0,Y 333.01,Z 729.885,A -85,B 0,C 180,E1 14931.839,E2 14931.839} C_VEL
LIN {X 0,Y 330.504,Z 727.048,A -85,B 0,C 180,E1 14940.662,E2 14940.662} C_VEL
LIN {X 0,Y 333.943,Z 731.062,A -85,B 0,C 180,E1 14948.643,E2 14948.643} C_VEL
LIN {X 0,Y 338.854,Z 739.277,A -85,B 0,C 180,E1 14953.983,E2 14953.983} C_VEL
LIN {X 0,Y 343.657,Z 746.945,A -85,B 0,C 180,E1 14957.636,E2 14957.636} C_VEL
LIN {X 0,Y 352.743,Z 761.859,A -85,B 0,C 180,E1 14963.171,E2 14963.171} C_VEL
LIN {X 0,Y 363.804,Z 784.743,A -85,B 0,C 180,E1 14969.076,E2 14969.076} C_VEL
LIN {X 0,Y 372.971,Z 809.01,A -85,B 0,C 180,E1 14973.932,E2 14973.932} C_VEL
LIN {X 0,Y 373.92,Z 814.989,A -85,B 0,C 180,E1 14974.833,E2 14974.833} C_VEL
LIN {X 0,Y 362.355,Z 854.371,A -85,B 0,C 180,E1 14977.694,E2 14977.694} C_VEL
LIN {X 0,Y 349.638,Z 890.192,A -85,B 0,C 180,E1 14981.436,E2 14981.436} C_VEL
LIN {X 0,Y 335.957,Z 923.96,A -85,B 0,C 180,E1 14986.382,E2 14986.382} C_VEL
LIN {X 0,Y 323.25,Z 953.657,A -85,B 0,C 180,E1 14992.49,E2 14992.49} C_VEL
LIN {X 0,Y 313.099,Z 977.98,A -85,B 0,C 180,E1 14999.486,E2 14999.486} C_VEL
LIN {X 0,Y 306.199,Z 997.373,A -85,B 0,C 180,E1 15007.467,E2 15007.467} C_VEL
LIN {X 0,Y 302.991,Z 1010.349,A -85,B 0,C 180,E1 15015.532,E2 15015.532} C_VEL
LIN {X 0,Y 302.138,Z 1016.126,A -85,B 0,C 180,E1 15021.354,E2 15021.354} C_VEL
LIN {X 0,Y 302.023,Z 1018.989,A -85,B 0,C 180,E1 15027.127,E2 15027.127} C_VEL
LIN {X 0,Y 301.954,Z 1018.987,A -85,B 0,C 180,E1 15032.875,E2 15032.875} C_VEL
LIN {X 0,Y 302.267,Z 1014.884,A -85,B 0,C 180,E1 15040.098,E2 15040.098} C_VEL
LIN {X 0,Y 303.829,Z 1006.328,A -85,B 0,C 180,E1 15047.398,E2 15047.398} C_VEL
LIN {X 0,Y 308.286,Z 991.108,A -85,B 0,C 180,E1 15055.472,E2 15055.472} C_VEL
LIN {X 0,Y 316.614,Z 969.307,A -85,B 0,C 180,E1 15063.302,E2 15063.302} C_VEL
LIN {X 0,Y 328.322,Z 941.805,A -85,B 0,C 180,E1 15070.213,E2 15070.213} C_VEL
LIN {X 0,Y 334.822,Z 926.631,A -85,B 0,C 180,E1 15073.147,E2 15073.147} C_VEL
LIN {X 0,Y 336.522,Z 915.666,A -85,B 0,C 180,E1 15075.469,E2 15075.469} C_VEL
LIN {X 0,Y 338.433,Z 904.157,A -85,B 0,C 180,E1 15077.693,E2 15077.693} C_VEL
LIN {X 0,Y 351.745,Z 870.491,A -85,B 0,C 180,E1 15081.774,E2 15081.774} C_VEL
LIN {X 0,Y 363.903,Z 834.629,A -85,B 0,C 180,E1 15084.871,E2 15084.871} C_VEL
LIN {X 0,Y 368.816,Z 816.844,A -85,B 0,C 180,E1 15086.082,E2 15086.082} C_VEL
LIN {X 0,Y 360.196,Z 791.789,A -85,B 0,C 180,E1 15091.201,E2 15091.201} C_VEL
LIN {X 0,Y 350.635,Z 770.887,A -85,B 0,C 180,E1 15096.649,E2 15096.649} C_VEL
LIN {X 0,Y 342.381,Z 755.965,A -85,B 0,C 180,E1 15101.964,E2 15101.964} C_VEL
LIN {X 0,Y 337.993,Z 748.86,A -85,B 0,C 180,E1 15105.401,E2 15105.401} C_VEL
LIN {X 0,Y 335.022,Z 743.877,A -85,B 0,C 180,E1 15108.261,E2 15108.261} C_VEL
LIN {X 0,Y 331.447,Z 737.484,A -85,B 0,C 180,E1 15113.108,E2 15113.108} C_VEL
LIN {X 0,Y 329.252,Z 735.213,A -85,B 0,C 180,E1 15121.311,E2 15121.311} C_VEL
LIN {X 0,Y 332.054,Z 738.813,A -85,B 0,C 180,E1 15128.762,E2 15128.762} C_VEL
LIN {X 0,Y 336.371,Z 746.726,A -85,B 0,C 180,E1 15134.159,E2 15134.159} C_VEL
LIN {X 0,Y 342.53,Z 757.375,A -85,B 0,C 180,E1 15139.352,E2 15139.352} C_VEL
LIN {X 0,Y 351.364,Z 775.681,A -85,B 0,C 180,E1 15145.515,E2 15145.515} C_VEL
LIN {X 0,Y 359.247,Z 795.865,A -85,B 0,C 180,E1 15150.657,E2 15150.657} C_VEL
LIN {X 0,Y 365.07,Z 817.167,A -85,B 0,C 180,E1 15155.109,E2 15155.109} C_VEL
LIN {X 0,Y 363.737,Z 823.644,A -85,B 0,C 180,E1 15155.742,E2 15155.742} C_VEL
LIN {X 0,Y 350.677,Z 861.169,A -85,B 0,C 180,E1 15159.267,E2 15159.267} C_VEL
LIN {X 0,Y 336.385,Z 895.811,A -85,B 0,C 180,E1 15163.931,E2 15163.931} C_VEL
LIN {X 0,Y 323.026,Z 924.923,A -85,B 0,C 180,E1 15169.431,E2 15169.431} C_VEL
LIN {X 0,Y 311.378,Z 949.293,A -85,B 0,C 180,E1 15175.87,E2 15175.87} C_VEL
LIN {X 0,Y 302.566,Z 968.96,A -85,B 0,C 180,E1 15183.232,E2 15183.232} C_VEL
LIN {X 0,Y 297.264,Z 983.322,A -85,B 0,C 180,E1 15191.097,E2 15191.097} C_VEL
LIN {X 0,Y 294.876,Z 991.721,A -85,B 0,C 180,E1 15198.147,E2 15198.147} C_VEL
LIN {X 0,Y 294.175,Z 995.696,A -85,B 0,C 180,E1 15204.091,E2 15204.091} C_VEL
LIN {X 0,Y 294.157,Z 996.989,A -85,B 0,C 180,E1 15209.999,E2 15209.999} C_VEL
LIN {X 0,Y 294.123,Z 995.654,A -85,B 0,C 180,E1 15215.909,E2 15215.909} C_VEL
LIN {X 0,Y 295.15,Z 990.477,A -85,B 0,C 180,E1 15222.988,E2 15222.988} C_VEL
LIN {X 0,Y 298.263,Z 980.246,A -85,B 0,C 180,E1 15230.814,E2 15230.814} C_VEL
LIN {X 0,Y 304.823,Z 963.602,A -85,B 0,C 180,E1 15238.965,E2 15238.965} C_VEL
LIN {X 0,Y 315.374,Z 941.02,A -85,B 0,C 180,E1 15246.449,E2 15246.449} C_VEL
LIN {X 0,Y 328.458,Z 913.18,A -85,B 0,C 180,E1 15252.908,E2 15252.908} C_VEL
LIN {X 0,Y 342.73,Z 880.793,A -85,B 0,C 180,E1 15258.201,E2 15258.201} C_VEL
LIN {X 0,Y 356.404,Z 845.609,A -85,B 0,C 180,E1 15262.246,E2 15262.246} C_VEL
LIN {X 0,Y 365.293,Z 818.479,A -85,B 0,C 180,E1 15264.543,E2 15264.543} C_VEL
LIN {X 0,Y 359.312,Z 796.336,A -85,B 0,C 180,E1 15269.133,E2 15269.133} C_VEL
LIN {X 0,Y 350.326,Z 773.373,A -85,B 0,C 180,E1 15275.02,E2 15275.02} C_VEL
LIN {X 0,Y 341.881,Z 756.388,A -85,B 0,C 180,E1 15280.946,E2 15280.946} C_VEL
LIN {X 0,Y 335.151,Z 744.243,A -85,B 0,C 180,E1 15286.954,E2 15286.954} C_VEL
LIN {X 0,Y 331.305,Z 737.522,A -85,B 0,C 180,E1 15292.127,E2 15292.127} C_VEL
LIN {X 0,Y 329.098,Z 734.827,A -85,B 0,C 180,E1 15300.665,E2 15300.665} C_VEL
LIN {X 0,Y 332.206,Z 738.652,A -85,B 0,C 180,E1 15308.358,E2 15308.358} C_VEL
LIN {X 0,Y 336.953,Z 746.888,A -85,B 0,C 180,E1 15313.732,E2 15313.732} C_VEL
LIN {X 0,Y 341.921,Z 755.331,A -85,B 0,C 180,E1 15317.811,E2 15317.811} C_VEL
LIN {X 0,Y 350.073,Z 769.818,A -85,B 0,C 180,E1 15323.075,E2 15323.075} C_VEL
LIN {X 0,Y 359.918,Z 791.204,A -85,B 0,C 180,E1 15328.694,E2 15328.694} C_VEL
LIN {X 0,Y 368.156,Z 814.876,A -85,B 0,C 180,E1 15333.556,E2 15333.556} C_VEL
LIN {X 0,Y 368.292,Z 818.861,A -85,B 0,C 180,E1 15334.067,E2 15334.067} C_VEL
LIN {X 0,Y 356.413,Z 857.161,A -85,B 0,C 180,E1 15336.949,E2 15336.949} C_VEL
LIN {X 0,Y 343.169,Z 892.516,A -85,B 0,C 180,E1 15340.747,E2 15340.747} C_VEL
LIN {X 0,Y 329.888,Z 923.952,A -85,B 0,C 180,E1 15345.448,E2 15345.448} C_VEL
LIN {X 0,Y 316.7,Z 953.343,A -85,B 0,C 180,E1 15351.574,E2 15351.574} C_VEL
LIN {X 0,Y 305.967,Z 977.667,A -85,B 0,C 180,E1 15358.696,E2 15358.696} C_VEL
LIN {X 0,Y 298.641,Z 997.064,A -85,B 0,C 180,E1 15366.864,E2 15366.864} C_VEL
LIN {X 0,Y 295.204,Z 1010.047,A -85,B 0,C 180,E1 15375.141,E2 15375.141} C_VEL
LIN {X 0,Y 294.245,Z 1015.826,A -85,B 0,C 180,E1 15381.12,E2 15381.12} C_VEL
LIN {X 0,Y 294.112,Z 1018.692,A -85,B 0,C 180,E1 15387.05,E2 15387.05} C_VEL
LIN {X 0,Y 294.046,Z 1018.691,A -85,B 0,C 180,E1 15392.952,E2 15392.952} C_VEL
LIN {X 0,Y 294.405,Z 1014.585,A -85,B 0,C 180,E1 15400.37,E2 15400.37} C_VEL
LIN {X 0,Y 296.089,Z 1006.024,A -85,B 0,C 180,E1 15407.868,E2 15407.868} C_VEL
LIN {X 0,Y 300.981,Z 990.575,A -85,B 0,C 180,E1 15416.244,E2 15416.244} C_VEL
LIN {X 0,Y 309.822,Z 968.803,A -85,B 0,C 180,E1 15424.198,E2 15424.198} C_VEL
LIN {X 0,Y 322.059,Z 941.498,A -85,B 0,C 180,E1 15431.162,E2 15431.162} C_VEL
LIN {X 0,Y 335.894,Z 910.452,A -85,B 0,C 180,E1 15436.759,E2 15436.759} C_VEL
LIN {X 0,Y 338.433,Z 904.157,A -85,B 0,C 180,E1 15437.693,E2 15437.693} C_VEL
LIN {X 0,Y 340.621,Z 892.152,A -85,B 0,C 180,E1 15439.826,E2 15439.826} C_VEL
LIN {X 0,Y 342.506,Z 881.3,A -85,B 0,C 180,E1 15441.612,E2 15441.612} C_VEL
LIN {X 0,Y 343.165,Z 879.584,A -85,B 0,C 180,E1 15441.814,E2 15441.814} C_VEL
LIN {X 0,Y 356.452,Z 842.996,A -85,B 0,C 180,E1 15445.277,E2 15445.277} C_VEL
LIN {X 0,Y 363.279,Z 820.145,A -85,B 0,C 180,E1 15446.943,E2 15446.943} C_VEL
LIN {X 0,Y 354.923,Z 794.796,A -85,B 0,C 180,E1 15452.373,E2 15452.373} C_VEL
LIN {X 0,Y 345.704,Z 774.123,A -85,B 0,C 180,E1 15458.152,E2 15458.152} C_VEL
LIN {X 0,Y 337.143,Z 758.001,A -85,B 0,C 180,E1 15464.531,E2 15464.531} C_VEL
LIN {X 0,Y 332.672,Z 751.021,A -85,B 0,C 180,E1 15468.842,E2 15468.842} C_VEL
LIN {X 0,Y 329.957,Z 745.239,A -85,B 0,C 180,E1 15473.076,E2 15473.076} C_VEL
LIN {X 0,Y 327.759,Z 742.968,A -85,B 0,C 180,E1 15481.317,E2 15481.317} C_VEL
LIN {X 0,Y 330.183,Z 746.451,A -85,B 0,C 180,E1 15488.563,E2 15488.563} C_VEL
LIN {X 0,Y 334.148,Z 754.194,A -85,B 0,C 180,E1 15493.889,E2 15493.889} C_VEL
LIN {X 0,Y 339.764,Z 764.764,A -85,B 0,C 180,E1 15499.093,E2 15499.093} C_VEL
LIN {X 0,Y 347.681,Z 782.055,A -85,B 0,C 180,E1 15505.049,E2 15505.049} C_VEL
LIN {X 0,Y 354.721,Z 801.764,A -85,B 0,C 180,E1 15510.224,E2 15510.224} C_VEL
LIN {X 0,Y 359.612,Z 822.526,A -85,B 0,C 180,E1 15514.598,E2 15514.598} C_VEL
LIN {X 0,Y 345.701,Z 861.341,A -85,B 0,C 180,E1 15518.221,E2 15518.221} C_VEL
LIN {X 0,Y 330.82,Z 896.111,A -85,B 0,C 180,E1 15522.921,E2 15522.921} C_VEL
LIN {X 0,Y 316.851,Z 925.227,A -85,B 0,C 180,E1 15528.469,E2 15528.469} C_VEL
LIN {X 0,Y 304.048,Z 950.822,A -85,B 0,C 180,E1 15535.396,E2 15535.396} C_VEL
LIN {X 0,Y 294.609,Z 970.984,A -85,B 0,C 180,E1 15543.305,E2 15543.305} C_VEL
LIN {X 0,Y 289.105,Z 985.229,A -85,B 0,C 180,E1 15551.685,E2 15551.685} C_VEL
LIN {X 0,Y 286.8,Z 993.19,A -85,B 0,C 180,E1 15559.352,E2 15559.352} C_VEL
LIN {X 0,Y 286.221,Z 996.969,A -85,B 0,C 180,E1 15566.967,E2 15566.967} C_VEL
LIN {X 0,Y 286.173,Z 996.95,A -85,B 0,C 180,E1 15573.032,E2 15573.032} C_VEL
LIN {X 0,Y 286.799,Z 993.116,A -85,B 0,C 180,E1 15580.647,E2 15580.647} C_VEL
LIN {X 0,Y 289.121,Z 985.09,A -85,B 0,C 180,E1 15588.313,E2 15588.313} C_VEL
LIN {X 0,Y 294.7,Z 970.748,A -85,B 0,C 180,E1 15596.711,E2 15596.711} C_VEL
LIN {X 0,Y 304.343,Z 950.294,A -85,B 0,C 180,E1 15604.67,E2 15604.67} C_VEL
LIN {X 0,Y 317.008,Z 924.885,A -85,B 0,C 180,E1 15611.505,E2 15611.505} C_VEL
LIN {X 0,Y 331.849,Z 893.733,A -85,B 0,C 180,E1 15617.367,E2 15617.367} C_VEL
LIN {X 0,Y 346.854,Z 858.383,A -85,B 0,C 180,E1 15621.995,E2 15621.995} C_VEL
LIN {X 0,Y 359.641,Z 821.087,A -85,B 0,C 180,E1 15625.504,E2 15625.504} C_VEL
LIN {X 0,Y 353.213,Z 797.286,A -85,B 0,C 180,E1 15630.757,E2 15630.757} C_VEL
LIN {X 0,Y 345.435,Z 777.137,A -85,B 0,C 180,E1 15636.343,E2 15636.343} C_VEL
LIN {X 0,Y 337.724,Z 761.3,A -85,B 0,C 180,E1 15642.356,E2 15642.356} C_VEL
LIN {X 0,Y 332.673,Z 751.416,A -85,B 0,C 180,E1 15647.523,E2 15647.523} C_VEL
LIN {X 0,Y 329.475,Z 745.118,A -85,B 0,C 180,E1 15652.415,E2 15652.415} C_VEL
LIN {X 0,Y 327.605,Z 742.585,A -85,B 0,C 180,E1 15660.668,E2 15660.668} C_VEL
LIN {X 0,Y 330.473,Z 746.402,A -85,B 0,C 180,E1 15668.154,E2 15668.154} C_VEL
LIN {X 0,Y 334.828,Z 754.536,A -85,B 0,C 180,E1 15673.571,E2 15673.571} C_VEL
LIN {X 0,Y 340.743,Z 764.572,A -85,B 0,C 180,E1 15678.44,E2 15678.44} C_VEL
LIN {X 0,Y 348.928,Z 781.07,A -85,B 0,C 180,E1 15684.008,E2 15684.008} C_VEL
LIN {X 0,Y 357.743,Z 802.674,A -85,B 0,C 180,E1 15689.475,E2 15689.475} C_VEL
LIN {X 0,Y 363.188,Z 820.148,A -85,B 0,C 180,E1 15693.063,E2 15693.063} C_VEL
LIN {X 0,Y 350.481,Z 859.95,A -85,B 0,C 180,E1 15696.168,E2 15696.168} C_VEL
LIN {X 0,Y 336.114,Z 896.427,A -85,B 0,C 180,E1 15700.244,E2 15700.244} C_VEL
LIN {X 0,Y 322.159,Z 927.709,A -85,B 0,C 180,E1 15705.174,E2 15705.174} C_VEL
LIN {X 0,Y 308.914,Z 955.81,A -85,B 0,C 180,E1 15711.349,E2 15711.349} C_VEL
LIN {X 0,Y 298.962,Z 977.356,A -85,B 0,C 180,E1 15717.876,E2 15717.876} C_VEL
LIN {X 0,Y 291.137,Z 996.757,A -85,B 0,C 180,E1 15726.232,E2 15726.232} C_VEL
LIN {X 0,Y 287.39,Z 1009.743,A -85,B 0,C 180,E1 15734.728,E2 15734.728} C_VEL
LIN {X 0,Y 286.361,Z 1015.526,A -85,B 0,C 180,E1 15740.874,E2 15740.874} C_VEL
LIN {X 0,Y 286.211,Z 1018.395,A -85,B 0,C 180,E1 15746.968,E2 15746.968} C_VEL
LIN {X 0,Y 286.156,Z 1018.395,A -85,B 0,C 180,E1 15753.034,E2 15753.034} C_VEL
LIN {X 0,Y 286.525,Z 1014.285,A -85,B 0,C 180,E1 15760.659,E2 15760.659} C_VEL
LIN {X 0,Y 288.366,Z 1005.721,A -85,B 0,C 180,E1 15768.363,E2 15768.363} C_VEL
LIN {X 0,Y 293.509,Z 990.536,A -85,B 0,C 180,E1 15776.832,E2 15776.832} C_VEL
LIN {X 0,Y 302.868,Z 968.854,A -85,B 0,C 180,E1 15784.969,E2 15784.969} C_VEL
LIN {X 0,Y 315.907,Z 941.191,A -85,B 0,C 180,E1 15792.145,E2 15792.145} C_VEL
LIN {X 0,Y 330.602,Z 909.348,A -85,B 0,C 180,E1 15797.927,E2 15797.927} C_VEL
LIN {X 0,Y 343.165,Z 879.584,A -85,B 0,C 180,E1 15801.814,E2 15801.814} C_VEL
LIN {X 0,Y 345.823,Z 866.518,A -85,B 0,C 180,E1 15803.705,E2 15803.705} C_VEL
LIN {X 0,Y 348.287,Z 853.031,A -85,B 0,C 180,E1 15805.513,E2 15805.513} C_VEL
LIN {X 0,Y 357.764,Z 823.487,A -85,B 0,C 180,E1 15807.825,E2 15807.825} C_VEL
LIN {X 0,Y 350.44,Z 800.136,A -85,B 0,C 180,E1 15813.019,E2 15813.019} C_VEL
LIN {X 0,Y 342.008,Z 780.083,A -85,B 0,C 180,E1 15818.855,E2 15818.855} C_VEL
LIN {X 0,Y 334.449,Z 765.086,A -85,B 0,C 180,E1 15824.991,E2 15824.991} C_VEL
LIN {X 0,Y 330.368,Z 758.211,A -85,B 0,C 180,E1 15829.308,E2 15829.308} C_VEL
LIN {X 0,Y 327.719,Z 752.698,A -85,B 0,C 180,E1 15833.695,E2 15833.695} C_VEL
LIN {X 0,Y 325.943,Z 750.64,A -85,B 0,C 180,E1 15841.324,E2 15841.324} C_VEL
LIN {X 0,Y 328.157,Z 754.006,A -85,B 0,C 180,E1 15848.317,E2 15848.317} C_VEL
LIN {X 0,Y 331.847,Z 761.953,A -85,B 0,C 180,E1 15853.84,E2 15853.84} C_VEL
LIN {X 0,Y 336.411,Z 770.817,A -85,B 0,C 180,E1 15858.355,E2 15858.355} C_VEL
LIN {X 0,Y 343.939,Z 788.709,A -85,B 0,C 180,E1 15864.711,E2 15864.711} C_VEL
LIN {X 0,Y 350.637,Z 809.294,A -85,B 0,C 180,E1 15870.156,E2 15870.156} C_VEL
LIN {X 0,Y 354.259,Z 825.374,A -85,B 0,C 180,E1 15873.74,E2 15873.74} C_VEL
LIN {X 0,Y 340.822,Z 861.636,A -85,B 0,C 180,E1 15877.168,E2 15877.168} C_VEL
LIN {X 0,Y 326.225,Z 894.69,A -85,B 0,C 180,E1 15881.596,E2 15881.596} C_VEL
LIN {X 0,Y 310.814,Z 925.529,A -85,B 0,C 180,E1 15887.475,E2 15887.475} C_VEL
LIN {X 0,Y 297.333,Z 951.223,A -85,B 0,C 180,E1 15894.54,E2 15894.54} C_VEL
LIN {X 0,Y 287.485,Z 971.008,A -85,B 0,C 180,E1 15902.435,E2 15902.435} C_VEL
LIN {X 0,Y 281.46,Z 985.531,A -85,B 0,C 180,E1 15911.169,E2 15911.169} C_VEL
LIN {X 0,Y 278.966,Z 993.489,A -85,B 0,C 180,E1 15919.049,E2 15919.049} C_VEL
LIN {X 0,Y 278.318,Z 997.266,A -85,B 0,C 180,E1 15926.881,E2 15926.881} C_VEL
LIN {X 0,Y 278.27,Z 997.247,A -85,B 0,C 180,E1 15933.118,E2 15933.118} C_VEL
LIN {X 0,Y 278.967,Z 993.415,A -85,B 0,C 180,E1 15940.95,E2 15940.95} C_VEL
LIN {X 0,Y 281.479,Z 985.393,A -85,B 0,C 180,E1 15948.828,E2 15948.828} C_VEL
LIN {X 0,Y 287.609,Z 970.784,A -85,B 0,C 180,E1 15957.564,E2 15957.564} C_VEL
LIN {X 0,Y 298.105,Z 949.876,A -85,B 0,C 180,E1 15965.78,E2 15965.78} C_VEL
LIN {X 0,Y 311.739,Z 923.633,A -85,B 0,C 180,E1 15972.84,E2 15972.84} C_VEL
LIN {X 0,Y 326.357,Z 894.149,A -85,B 0,C 180,E1 15978.399,E2 15978.399} C_VEL
LIN {X 0,Y 341.973,Z 858.689,A -85,B 0,C 180,E1 15983.054,E2 15983.054} C_VEL
LIN {X 0,Y 354.162,Z 824.865,A -85,B 0,C 180,E1 15986.249,E2 15986.249} C_VEL
LIN {X 0,Y 348.459,Z 802.234,A -85,B 0,C 180,E1 15991.459,E2 15991.459} C_VEL
LIN {X 0,Y 341.566,Z 782.784,A -85,B 0,C 180,E1 15997.058,E2 15997.058} C_VEL
LIN {X 0,Y 333.515,Z 764.941,A -85,B 0,C 180,E1 16004.202,E2 16004.202} C_VEL
LIN {X 0,Y 329.979,Z 758.373,A -85,B 0,C 180,E1 16008.26,E2 16008.26} C_VEL
LIN {X 0,Y 327.458,Z 752.647,A -85,B 0,C 180,E1 16012.702,E2 16012.702} C_VEL
LIN {X 0,Y 325.82,Z 750.286,A -85,B 0,C 180,E1 16020.672,E2 16020.672} C_VEL
LIN {X 0,Y 328.448,Z 754.04,A -85,B 0,C 180,E1 16027.954,E2 16027.954} C_VEL
LIN {X 0,Y 332.533,Z 761.829,A -85,B 0,C 180,E1 16033.248,E2 16033.248} C_VEL
LIN {X 0,Y 338.07,Z 772.233,A -85,B 0,C 180,E1 16038.274,E2 16038.274} C_VEL
LIN {X 0,Y 345.426,Z 787.876,A -85,B 0,C 180,E1 16043.657,E2 16043.657} C_VEL
LIN {X 0,Y 353.433,Z 808.742,A -85,B 0,C 180,E1 16049.049,E2 16049.049} C_VEL
LIN {X 0,Y 357.639,Z 824.75,A -85,B 0,C 180,E1 16052.356,E2 16052.356} C_VEL
LIN {X 0,Y 344.091,Z 864.137,A -85,B 0,C 180,E1 16055.508,E2 16055.508} C_VEL
LIN {X 0,Y 328.684,Z 901.102,A -85,B 0,C 180,E1 16059.839,E2 16059.839} C_VEL
LIN {X 0,Y 313.856,Z 932.695,A -85,B 0,C 180,E1 16065.128,E2 16065.128} C_VEL
LIN {X 0,Y 299.844,Z 960.864,A -85,B 0,C 180,E1 16071.813,E2 16071.813} C_VEL
LIN {X 0,Y 289.039,Z 983.656,A -85,B 0,C 180,E1 16079.563,E2 16079.563} C_VEL
LIN {X 0,Y 282.178,Z 1000.582,A -85,B 0,C 180,E1 16087.939,E2 16087.939} C_VEL
LIN {X 0,Y 279.181,Z 1011.088,A -85,B 0,C 180,E1 16095.875,E2 16095.875} C_VEL
LIN {X 0,Y 278.248,Z 1017.019,A -85,B 0,C 180,E1 16103.753,E2 16103.753} C_VEL
LIN {X 0,Y 278.42,Z 1018.462,A -85,B 0,C 180,E1 16110.001,E2 16110.001} C_VEL
LIN {X 0,Y 278.249,Z 1017.022,A -85,B 0,C 180,E1 16116.248,E2 16116.248} C_VEL
LIN {X 0,Y 279.182,Z 1011.095,A -85,B 0,C 180,E1 16124.126,E2 16124.126} C_VEL
LIN {X 0,Y 282.159,Z 1000.598,A -85,B 0,C 180,E1 16132.064,E2 16132.064} C_VEL
LIN {X 0,Y 288.912,Z 984.021,A -85,B 0,C 180,E1 16140.288,E2 16140.288} C_VEL
LIN {X 0,Y 300.43,Z 959.677,A -85,B 0,C 180,E1 16148.53,E2 16148.53} C_VEL
LIN {X 0,Y 314.701,Z 931.021,A -85,B 0,C 180,E1 16155.207,E2 16155.207} C_VEL
LIN {X 0,Y 330.022,Z 898.272,A -85,B 0,C 180,E1 16160.565,E2 16160.565} C_VEL
LIN {X 0,Y 345.271,Z 861.344,A -85,B 0,C 180,E1 16164.761,E2 16164.761} C_VEL
LIN {X 0,Y 348.287,Z 853.031,A -85,B 0,C 180,E1 16165.513,E2 16165.513} C_VEL
LIN {X 0,Y 349.259,Z 844.152,A -85,B 0,C 180,E1 16166.802,E2 16166.802} C_VEL
LIN {X 0,Y 350.17,Z 834.984,A -85,B 0,C 180,E1 16168.014,E2 16168.014} C_VEL
LIN {X 0,Y 352.391,Z 827.316,A -85,B 0,C 180,E1 16168.601,E2 16168.601} C_VEL
LIN {X 0,Y 345.542,Z 804.23,A -85,B 0,C 180,E1 16174.01,E2 16174.01} C_VEL
LIN {X 0,Y 338.333,Z 786.144,A -85,B 0,C 180,E1 16179.484,E2 16179.484} C_VEL
LIN {X 0,Y 331.595,Z 772.066,A -85,B 0,C 180,E1 16185.472,E2 16185.472} C_VEL
LIN {X 0,Y 328.054,Z 765.682,A -85,B 0,C 180,E1 16189.524,E2 16189.524} C_VEL
LIN {X 0,Y 325.86,Z 760.387,A -85,B 0,C 180,E1 16193.659,E2 16193.659} C_VEL
LIN {X 0,Y 324.094,Z 758.309,A -85,B 0,C 180,E1 16201.332,E2 16201.332} C_VEL
LIN {X 0,Y 325.932,Z 761.533,A -85,B 0,C 180,E1 16208.096,E2 16208.096} C_VEL
LIN {X 0,Y 329.106,Z 768.758,A -85,B 0,C 180,E1 16213.29,E2 16213.29} C_VEL
LIN {X 0,Y 335.327,Z 782.56,A -85,B 0,C 180,E1 16219.939,E2 16219.939} C_VEL
LIN {X 0,Y 342.27,Z 801.657,A -85,B 0,C 180,E1 16226.244,E2 16226.244} C_VEL
LIN {X 0,Y 347.633,Z 822.646,A -85,B 0,C 180,E1 16231.498,E2 16231.498} C_VEL
LIN {X 0,Y 348.365,Z 829.945,A -85,B 0,C 180,E1 16232.99,E2 16232.99} C_VEL
LIN {X 0,Y 334.337,Z 865.686,A -85,B 0,C 180,E1 16236.502,E2 16236.502} C_VEL
LIN {X 0,Y 319.439,Z 897.849,A -85,B 0,C 180,E1 16240.991,E2 16240.991} C_VEL
LIN {X 0,Y 304.043,Z 927.265,A -85,B 0,C 180,E1 16246.785,E2 16246.785} C_VEL
LIN {X 0,Y 290.745,Z 951.526,A -85,B 0,C 180,E1 16253.61,E2 16253.61} C_VEL
LIN {X 0,Y 280.142,Z 971.54,A -85,B 0,C 180,E1 16261.776,E2 16261.776} C_VEL
LIN {X 0,Y 273.818,Z 985.833,A -85,B 0,C 180,E1 16270.623,E2 16270.623} C_VEL
LIN {X 0,Y 271.118,Z 993.843,A -85,B 0,C 180,E1 16278.805,E2 16278.805} C_VEL
LIN {X 0,Y 270.419,Z 997.563,A -85,B 0,C 180,E1 16286.79,E2 16286.79} C_VEL
LIN {X 0,Y 270.376,Z 997.544,A -85,B 0,C 180,E1 16293.21,E2 16293.21} C_VEL
LIN {X 0,Y 271.12,Z 993.767,A -85,B 0,C 180,E1 16301.199,E2 16301.199} C_VEL
LIN {X 0,Y 273.849,Z 985.697,A -85,B 0,C 180,E1 16309.373,E2 16309.373} C_VEL
LIN {X 0,Y 280.271,Z 971.354,A -85,B 0,C 180,E1 16318.209,E2 16318.209} C_VEL
LIN {X 0,Y 291.175,Z 950.868,A -85,B 0,C 180,E1 16326.498,E2 16326.498} C_VEL
LIN {X 0,Y 305.014,Z 925.5,A -85,B 0,C 180,E1 16333.531,E2 16333.531} C_VEL
LIN {X 0,Y 320.919,Z 894.698,A -85,B 0,C 180,E1 16339.443,E2 16339.443} C_VEL
LIN {X 0,Y 337.23,Z 858.984,A -85,B 0,C 180,E1 16344.141,E2 16344.141} C_VEL
LIN {X 0,Y 348.631,Z 828.145,A -85,B 0,C 180,E1 16347.128,E2 16347.128} C_VEL
LIN {X 0,Y 343.469,Z 806.198,A -85,B 0,C 180,E1 16352.438,E2 16352.438} C_VEL
LIN {X 0,Y 337.005,Z 787.031,A -85,B 0,C 180,E1 16358.254,E2 16358.254} C_VEL
LIN {X 0,Y 330.362,Z 771.508,A -85,B 0,C 180,E1 16364.928,E2 16364.928} C_VEL
LIN {X 0,Y 327.3,Z 765.346,A -85,B 0,C 180,E1 16368.839,E2 16368.839} C_VEL
LIN {X 0,Y 325.293,Z 760.185,A -85,B 0,C 180,E1 16372.989,E2 16372.989} C_VEL
LIN {X 0,Y 323.98,Z 757.959,A -85,B 0,C 180,E1 16380.676,E2 16380.676} C_VEL
LIN {X 0,Y 326.367,Z 761.626,A -85,B 0,C 180,E1 16387.754,E2 16387.754} C_VEL
LIN {X 0,Y 330.14,Z 769.566,A -85,B 0,C 180,E1 16393.179,E2 16393.179} C_VEL
LIN {X 0,Y 335.139,Z 779.404,A -85,B 0,C 180,E1 16397.964,E2 16397.964} C_VEL
LIN {X 0,Y 342.075,Z 795.205,A -85,B 0,C 180,E1 16403.479,E2 16403.479} C_VEL
